Yaskawa INFORM job: X2_103(30,90)_V2.JBI

/JOB
//NAME X2_103(30,90)_V2
//POS
///NPOS 560,560,560,21,0,0
///TOOL 0
///POSTYPE PULSE
///PULSE
C00000=3271,-119374,-120746,-350,28955,423
C00001=-140235,-154096,-123138,2898,12995,-682
C00002=-200060,-156091,-101839,15852,59862,-55345
C00003=-224418,-53337,-27640,-2214,78542,-35069
C00004=-224438,-48029,-16239,-2251,74255,-34999
C00005=-222894,-44537,-9885,-2258,72183,-34438
C00006=-222281,-43062,-7261,-2261,71343,-34215
C00007=-219801,-41941,-6326,-2232,71409,-33379
C00008=-219801,-41166,-4818,-2238,70878,-33369
C00009=-219801,-41941,-6326,-2232,71409,-33379
C00010=-221729,-42672,-6756,-2255,71247,-34028
C00011=-221606,-41865,-5246,-2258,70739,-33978
C00012=-220679,-41360,-4730,-2248,70703,-33665
C00013=-221121,-41526,-4828,-2254,70667,-33813
C00014=-222894,-44537,-9885,-2258,72183,-34438
C00015=-224438,-48029,-16239,-2251,74255,-34999
C00016=-224391,-58970,-41460,-2187,84149,-35159
C00017=-200676,-32931,-16327,-317,66839,-14722
C00018=-188142,840,19554,1763,51642,-2042
C00019=-188000,8373,29094,1754,49640,-2018
C00020=-187946,11534,33150,1753,48768,-2011
C00021=-187952,12994,36316,1788,47570,-2035
C00022=-187946,11534,33150,1753,48768,-2011
C00023=-185876,12386,34874,-2226,48172,1956
C00024=-184694,15261,37512,-5775,48427,5518
C00025=-187925,12395,34881,1761,48145,-2013
C00026=-187893,12200,34611,1745,48210,-1998
C00027=-186938,14194,36446,1333,48088,-1587
C00028=-187893,12200,34611,1745,48210,-1998
C00029=-187946,9000,30501,1745,49095,-2005
C00030=-188087,1386,20853,1753,51122,-2028
C00031=-181732,-4900,4438,-770,58086,538
C00032=-174031,-1565,13615,-3944,54266,3743
C00033=-174319,5596,22673,-3924,52362,3698
C00034=-174429,8580,26495,-3922,51540,3684
C00035=-174433,9836,29416,-3983,50391,3728
C00036=-174429,8580,26495,-3922,51540,3684
C00037=-171116,10926,29585,-10065,52158,10061
C00038=-171940,12922,31394,-9974,52039,9961
C00039=-174482,9161,28010,-3935,50905,3687
C00040=-174468,9090,27852,-3937,50966,3690
C00041=-173667,11408,29941,-4272,50912,4030
C00042=-174468,9090,27852,-3937,50966,3690
C00043=-174358,6073,23987,-3937,51798,3704
C00044=-174072,-1158,14840,-3954,53720,3748
C00045=-173402,-7254,1011,1102,53334,3695
C00046=-173128,11811,16147,-4053,59614,3903
C00047=-173414,18752,25429,-4036,57459,3871
C00048=-173524,21666,29357,-4035,56536,3862
C00049=-173528,22669,32063,-4087,55389,3904
C00050=-173524,21666,29357,-4035,56536,3862
C00051=-172107,23003,31802,-6738,56186,6669
C00052=-172603,25249,33980,-7141,56088,7090
C00053=-173534,22315,31141,-4067,55773,3887
C00054=-175831,15088,24311,-3157,56159,2953
C00055=-175704,15840,26859,-3250,54984,3039
C00056=-174934,18176,29047,-3559,54871,3355
C00057=-175704,15840,26859,-3250,54984,3039
C00058=-175831,15088,24311,-3157,56159,2953
C00059=-173128,11811,16147,-4053,59614,3903
C00060=-158515,-47697,-14966,-51437,42315,-4350
C00061=-160188,-28820,10706,-61150,35121,-4094
C00062=-160938,-21306,18376,-62092,34254,-3699
C00063=-161219,-18227,21598,-62564,33894,-3488
C00064=-160407,-15938,23271,-62524,34443,-3379
C00065=-161219,-18227,21598,-62564,33894,-3488
C00066=-160594,-16595,22837,-62582,34299,-3378
C00067=-160592,-14820,26146,-64075,33771,-2570
C00068=-160594,-16595,22837,-62582,34299,-3378
C00069=-158698,-15537,23539,-63423,38355,-1788
C00070=-159328,-13237,25258,-63387,39000,-1639
C00071=-161141,-18339,21498,-62573,33942,-3471
C00072=-160858,-21416,18279,-62104,34303,-3680
C00073=-160103,-28926,10617,-61167,35171,-4072
C00074=-155148,-57735,-20992,-34211,37115,-7304
C00075=-144375,-92197,-43920,10369,38826,-10763
C00076=-123336,-72493,-22760,45909,48339,-7168
C00077=-110382,-36118,14049,67828,50364,-5484
C00078=-108060,-29324,20980,68768,48684,-5556
C00079=-107188,-26521,23897,69189,48032,-5626
C00080=-107504,-24071,25534,68933,48315,-5530
C00081=-107188,-26521,23897,69189,48032,-5626
C00082=-107470,-24738,25138,69020,48257,-5582
C00083=-107461,-22674,28687,69966,47830,-6220
C00084=-107470,-24738,25138,69020,48257,-5582
C00085=-107297,-26582,23837,69168,48098,-5639
C00086=-105452,-26141,24117,69389,47026,-5331
C00087=-107297,-26582,23837,69168,48098,-5639
C00088=-108171,-29382,20923,68748,48751,-5570
C00089=-110499,-36171,13998,67809,50435,-5499
C00090=-121659,-48497,-1187,64920,67113,80
C00091=-111034,-19450,-2794,41225,71575,-4827
C00092=-95590,24468,20339,13593,66440,-13992
C00093=-94636,30658,29262,13540,64031,-13917
C00094=-94266,33287,33052,13536,63014,-13897
C00095=-94260,34102,35593,13669,61899,-14031
C00096=-94266,33287,33052,13536,63014,-13897
C00097=-94257,33804,34719,13622,62273,-13984
C00098=-93260,34925,35856,13322,61987,-13631
C00099=-94257,33804,34719,13622,62273,-13984
C00100=-93131,24579,25521,13160,62983,-13463
C00101=-93277,25237,27975,13342,61865,-13653
C00102=-93655,28227,30921,13496,61658,-13825
C00103=-93277,25237,27975,13342,61865,-13653
C00104=-93131,24579,25521,13160,62983,-13463
C00105=-94266,33287,33052,13536,63014,-13897
C00106=-94636,30658,29262,13540,64031,-13917
C00107=-95590,24468,20339,13593,66440,-13992
C00108=-97908,6855,5922,13137,61050,-15522
C00109=-95297,11242,18824,14178,60690,-14590
C00110=-94266,17792,27740,14146,58451,-14474
C00111=-93867,20555,31520,14152,57502,-14440
C00112=-93860,21684,34363,14333,56366,-14591
C00113=-93867,20555,31520,14152,57502,-14440
C00114=-93834,21021,32943,14240,56879,-14511
C00115=-92751,22112,33981,13895,56618,-14106
C00116=-93834,21021,32943,14240,56879,-14511
C00117=-93847,20969,32801,14234,56940,-14507
C00118=-94233,23977,35706,14399,56772,-14687
C00119=-93847,20969,32801,14234,56940,-14507
C00120=-94245,18170,28975,14223,57899,-14539
C00121=-95277,11545,19966,14246,60155,-14652
C00122=-94527,-29265,-13111,13981,59468,-14364
C00123=-81565,-27458,3058,10852,48627,-10401
C00124=-80654,-20498,11026,10706,47205,-10165
C00125=-80308,-17644,14351,10663,46591,-10083
C00126=-80298,-16160,17342,10850,45531,-10203
C00127=-80308,-17644,14351,10663,46591,-10083
C00128=-80310,-16770,15973,10760,46052,-10147
C00129=-78983,-15416,16967,10190,45971,-9563
C00130=-80310,-16770,15973,10760,46052,-10147
C00131=-80369,-16920,15767,10776,46108,-10166
C00132=-81126,-14569,17524,11066,46330,-10477
C00133=-80369,-16920,15767,10776,46108,-10166
C00134=-80716,-19796,12409,10816,46731,-10247
C00135=-81629,-26799,4373,10955,48172,-10481
C00136=-81629,-36021,-16280,9851,56019,-9665
C00137=-81629,-36021,-16280,9851,56019,-9665
C00138=-81018,-22368,15352,11535,43694,-10760
C00139=-82220,-12770,25334,12334,42674,-11455
C00140=-82220,-11619,27495,12508,41954,-11560
C00141=-82220,-11847,27069,12473,42095,-11540
C00142=-82921,-9583,28807,12754,42287,-11838
C00143=-82839,-9854,28597,12721,42264,-11802
C00144=-82839,-10288,27783,12653,42536,-11762
C00145=-82987,-9794,28166,12713,42576,-11825
C00146=-82987,-9519,28676,12758,42403,-11847
C00147=-82987,-9667,28396,12734,42496,-11833
C00148=-83090,-9325,28661,12774,42522,-11877
C00149=-82753,-11045,26659,12547,42813,-11678
C00150=-119816,-37733,5380,24735,50291,-26788
C00151=-118732,-28444,14282,24759,49358,-26561
C00152=-118732,-27369,16233,24992,48768,-26724
C00153=-118733,-27539,15928,24955,48860,-26698
C00154=-118781,-24844,17728,24865,49124,-26646
C00155=-118771,-25424,17338,24885,49069,-26656
C00156=-118771,-25846,16569,24792,49302,-26592
C00157=-118785,-25058,17100,24768,49376,-26577
C00158=-118785,-24858,17464,24811,49265,-26606
C00159=-118785,-24952,17291,24791,49318,-26592
C00160=-118793,-24494,17602,24777,49360,-26584
C00161=-118763,-26610,15508,24704,49533,-26524
C00162=-155285,-26516,12514,28456,62214,-38311
C00163=-152438,-18325,21238,28659,60298,-37701
C00164=-152440,-17188,23354,28851,59667,-37879
C00165=-152440,-17414,22937,28813,59790,-37845
C00166=-151830,-15112,24623,28749,59726,-37617
C00167=-151901,-15387,24419,28758,59733,-37642
C00168=-151901,-15814,23624,28683,59971,-37576
C00169=-151771,-15314,23995,28670,59956,-37527
C00170=-151769,-15045,24491,28721,59807,-37565
C00171=-151767,-15191,24216,28696,59889,-37542
C00172=-151679,-14843,24474,28688,59877,-37510
C00173=-151971,-16573,22523,28616,60244,-37525
C00174=-150216,-29821,9901,28279,60539,-36735
C00175=-129415,-40611,3678,-20754,45854,21846
C00176=-132229,-30881,12703,-20034,44681,20835
C00177=-132233,-29758,14737,-20264,44044,20982
C00178=-132233,-29979,14337,-20217,44170,20950
C00179=-131980,-27625,15872,-20209,44476,20997
C00180=-132007,-27902,15689,-20213,44443,20995
C00181=-132009,-28325,14925,-20124,44681,20937
C00182=-131956,-27813,15263,-20122,44745,20946
C00183=-131946,-27551,15737,-20184,44594,20990
C00184=-131944,-27692,15476,-20156,44679,20973
C00185=-131906,-27334,15713,-20158,44724,20979
C00186=-132026,-29082,13878,-20039,44914,20879
C00187=-163713,-23600,14498,-6442,42405,6672
C00188=-163955,-12441,25582,-6447,41301,6644
C00189=-163960,-11291,27745,-6536,40565,6698
C00190=-163959,-11518,27319,-6518,40711,6685
C00191=-163182,-9327,29005,-6883,40857,7042
C00192=-163270,-9587,28803,-6845,40841,7005
C00193=-163272,-10021,27989,-6806,41118,6980
C00194=-163107,-9544,28360,-6883,41148,7055
C00195=-163099,-9280,28861,-6910,40971,7077
C00196=-163096,-9426,28582,-6901,41068,7072
C00197=-162981,-9093,28842,-6958,41088,7124
C00198=-163354,-10779,26863,-6731,41408,6921
C00199=-188135,19294,49745,5326,42598,-4607
C00200=-187094,34022,67542,5190,39163,-4331
C00201=-187099,35860,70809,5317,38103,-4403
C00202=-187098,35492,70157,5290,38315,-4390
C00203=-186242,38033,72879,4886,37897,-3996
C00204=-186340,37725,72546,4929,37948,-4039
C00205=-186342,37004,71278,4886,38357,-4015
C00206=-186159,37561,71878,4800,38266,-3932
C00207=-186153,37998,72654,4828,38007,-3942
C00208=-186151,37748,72215,4808,38149,-3930
C00209=-186023,38140,72638,4745,38082,-3873
C00210=-186437,35890,69530,4881,38858,-4029
C00211=-129415,-40611,3678,-20754,45854,21846
C00212=-138780,-33942,5724,-2673,47750,14957
C00213=-138299,-28814,11765,-2887,46684,15190
C00214=-170916,-2456,31220,8184,49299,1571
C00215=-171700,-5880,26786,8312,50334,1335
C00216=-135165,-49074,-6503,-3925,47635,16482
C00217=-161317,-13185,16777,20608,75826,-36642
C00218=-153104,-7651,23168,21233,72811,-34265
C00219=-161765,5352,36611,20811,73420,-37224
C00220=-160783,10050,41998,20985,72342,-37069
C00221=-152064,364,33603,21550,70406,-34339
C00222=-119342,-11748,23912,21569,62025,-23940
C00223=-119305,-17523,16883,21319,63284,-23678
C00224=-135165,-49074,-6503,-3925,47635,16482
C00225=-129415,-40611,3678,-20754,45854,21846
C00226=-171396,-8104,23990,8148,50880,1508
C00227=-170916,-2456,31220,8184,49299,1571
C00228=-192273,66939,103329,16264,43671,-8278
C00229=-192892,57382,88980,15390,47553,-7857
C00230=-135165,-49074,-6503,-3925,47635,16482
C00231=-161317,-13185,16777,20608,75826,-36642
C00232=-119244,-24750,9342,21153,64138,-23490
C00233=-119300,-17410,17676,21394,62882,-23755
C00234=-119342,-11748,23912,21569,62025,-23940
C00235=-84728,5286,37848,17156,54382,-11867
C00236=-85414,851,32833,17125,55288,-11988
C00237=-135165,-49074,-6503,-3925,47635,16482
C00238=-129360,-40332,3441,-20673,46138,21804
C00239=-138676,-33640,5524,-2697,48031,14993
C00240=-138191,-28354,11811,-2916,46896,15229
C00241=-170671,-2058,31280,8087,49442,1685
C00242=-171477,-5655,26582,8215,50551,1445
C00243=-135070,-48777,-6734,-3939,47933,16510
C00244=-161130,-12883,16630,20602,76011,-36544
C00245=-160264,65,29057,20749,74872,-36438
C00246=-160370,4102,35147,20897,73330,-36750
C00247=-164437,-245,35228,27243,65873,-40715
C00248=-155010,-10107,27390,27339,62790,-37870
C00249=-119242,-19669,19375,23179,54823,-25430
C00250=-119312,-17166,16760,21274,63528,-23633
C00251=-135070,-48777,-6734,-3939,47933,16510
C00252=-129360,-40332,3441,-20673,46138,21804
C00253=-171172,-7872,23791,8052,51098,1618
C00254=-170796,-1768,31531,8129,49447,1635
C00255=-192018,67019,103005,16124,43862,-8129
C00256=-192674,57393,88583,15275,47758,-7731
C00257=-135070,-48777,-6734,-3939,47933,16510
C00258=-161130,-12883,16630,20602,76011,-36544
C00259=-119252,-24388,9211,21109,64389,-23445
C00260=-119307,-17059,17547,21348,63127,-23710
C00261=-115642,-27884,15061,20579,45940,-25049
C00262=-76385,-6634,29757,2420,43140,-7452
C00263=-85568,1158,32706,17108,55544,-12007
C00264=-135070,-48777,-6734,-3939,47933,16510
C00265=-81018,-22368,15352,11535,43694,-10760
C00266=-90296,-130023,-32460,1589,43332,9709
C00267=-104076,-127604,-31640,1030,44224,5222
C00268=-104076,-125902,-29753,1035,43937,5219
C00269=-104076,-127604,-31640,1030,44224,5222
C00270=-75365,-129597,-31294,2148,42603,14582
C00271=-79043,-127585,-29221,2027,42422,13375
C00272=-98067,-126626,-29482,1288,43342,7171
C00273=-91643,-127131,-29393,1548,42950,9262
C00274=-91643,-133346,-36144,1521,43911,9279
C00275=-90543,-138207,-41193,1547,44504,9649
C00276=-97075,-139435,-37667,8780,42441,4238
C00277=-97192,-133417,-31365,8906,41673,4121
C00278=-82208,-129108,-27879,9651,40633,8927
C00279=-74453,-129099,-27873,9918,40030,11450
C00280=-77506,-125561,-24368,25333,36038,-6444
C00281=-97622,-127372,-24807,30901,38923,-18802
C00282=-97583,-132582,-30437,30417,39596,-18508
C00283=-96835,-139510,-37769,-4213,44951,10151
C00284=-96981,-133489,-31463,-4286,44162,10144
C00285=-62865,-129479,-28052,-642,44803,20513
C00286=-78696,-129496,-28185,-2375,44685,15709
C00287=-65731,-129649,-28076,-960,44711,19643
C00288=-97517,-133431,-31347,-4343,44102,9982
C00289=-97378,-139453,-37655,-4269,44892,9987
C00290=-122537,-139380,-37444,-6562,43692,2224
C00291=-122537,-133356,-31132,-6657,42908,2284
C00292=-123909,-129354,-27957,-6756,42937,1849
C00293=-136767,-129599,-28086,-7733,42151,-2168
C00294=-136042,-129584,-28096,-7681,42205,-1941
C00295=-122565,-109770,-4675,-55538,56258,9899
C00296=-122572,-114852,-10615,-54984,56869,9434
C00297=-218346,-133610,-69952,-6045,59781,-31164
C00298=-223401,-45840,-13156,-5364,69548,-33408
C00299=-222109,-41719,-6333,-5495,67560,-32869
C00300=-220997,-38818,-2909,-5568,67023,-32457
C00301=-222242,-31345,1911,-5480,67806,-32926
C00302=-220920,-39606,-2024,-7766,59138,-23574
C00303=-220403,-51511,-7368,-9623,49930,-15864
C00304=-221089,-58034,-14727,-9279,51017,-16249
C00305=-225149,-36583,-7538,-3060,79587,-35998
C00306=-223778,-33707,-1346,-2977,77308,-35487
C00307=-222503,-31636,1503,-2884,76662,-35050
C00308=-221605,-36907,-1779,-2822,76007,-34739
C00309=-217292,-55512,-12105,-2514,72937,-33253
C00310=-219328,-56399,-14375,-2668,73818,-33940
C00311=-221046,-59770,-20585,-2780,75851,-34551
C00312=-232710,-104201,-36509,-3988,62401,-37975
C00313=-229171,-99745,-30242,-3753,60982,-36787
C00314=-225249,-97366,-27202,-3443,60481,-35515
C00315=-159716,-121406,-28671,3019,49335,-15001
C00316=-178146,-119749,-28353,3122,51852,-21289
C00317=-201053,-127933,-48461,1469,67517,-27836
C00318=-218346,-133610,-69952,-6045,59781,-31164
C00319=-155907,-158824,-62139,3482,48253,-13777
C00320=-122507,-139290,-37311,6932,43923,-3746
C00321=-122509,-133268,-31001,7032,43139,-3809
C00322=-129091,-129141,-27877,6412,43686,-5823
C00323=-103454,-129456,-28220,8487,42206,2149
C00324=-122587,-133369,-31211,7015,43220,-3827
C00325=-122586,-139389,-37517,6916,44002,-3765
C00326=-178554,-156416,-68062,-1714,49894,-19175
C00327=-213759,-120199,-38675,-7265,47820,-28777
C00328=-208805,-113975,-32275,-7533,47440,-26995
C00329=-203457,-110659,-29180,-7720,47634,-25130
C00330=-226422,-78834,-22033,-5752,57916,-33897
C00331=-229015,-79900,-24597,-5554,58778,-34856
C00332=-231182,-84689,-31124,-5352,60195,-35689
C00333=-212528,-138829,-62774,-5865,50017,-28724
C00334=-155907,-158824,-62139,3482,48253,-13777
C00335=-121094,-142626,-31574,-10098,25521,4701
C00336=-121096,-137018,-25859,-10336,24895,4818
C00337=-164582,-134101,-22446,3427,23155,-15265
C00338=-111553,-133057,-22885,-12578,25881,8893
C00339=-110779,-133123,-22850,-12777,25898,9232
C00340=-112921,-147420,-34515,-12366,25547,8360
C00341=-112921,-149481,-36511,-12292,25712,8323
C00342=-97228,-139073,-37279,8780,42400,4184
C00343=-97344,-133056,-30967,8907,41624,4066
C00344=-78012,-130084,-28544,9824,40218,10278
C00345=-81788,-129487,-28074,9683,40529,9053
C00346=-82179,-129411,-27981,9668,40535,8924
C00347=-74028,-129648,-28142,9954,39883,11573
C00348=-97200,-133072,-30998,8914,41625,4113
C00349=-97082,-139088,-37310,8787,42400,4232
C00350=-94488,-144762,-30508,4018,22458,6207
C00351=-94506,-139089,-24810,4127,21868,6148
C00352=-109156,-134471,-22107,8848,23225,-653
C00353=-92905,-135418,-22246,3518,22151,6937
C00354=-86752,-134662,-22676,6773,23151,2299
C00355=-94482,-131728,-17188,50151,23285,-24299
C00356=-94477,-136650,-22327,49039,23703,-23756
C00357=-194092,-153326,-35489,27084,38346,-44238
C00358=-219173,-157061,-72685,-6819,49419,-30815
C00359=-224435,-92754,-33276,-5864,57810,-33193
C00360=-222031,-87567,-26717,-6069,56604,-32279
C00361=-219894,-84961,-24547,-6166,56749,-31533
C00362=-220391,-83143,-23447,-6127,56973,-31723
C00363=-220808,-82168,-23250,-6081,57322,-31890
C00364=-221831,-79477,-22462,-5978,58145,-32293
C00365=-223925,-82065,-24949,-5866,58209,-33035
C00366=-226120,-87049,-31520,-5671,59544,-33877
C00367=-225186,-114904,-34894,11668,45054,-37894
C00368=-216822,-109183,-29035,10924,43485,-34913
C00369=-213756,-104039,-26334,10373,44131,-33658
C00370=-227756,-76443,-19510,10264,55464,-37669
C00371=-223895,-83934,-20074,8254,42953,-29929
C00372=-217578,-99941,-27704,3828,33118,-22325
C00373=-218675,-113856,-37596,3440,30409,-21358
C00374=-233993,-86215,-29007,10771,66078,-41518
C00375=-229810,-82565,-23340,11182,63991,-40325
C00376=-227706,-76286,-19097,11255,64337,-39587
C00377=-202149,-109903,-26387,14167,48571,-32832
C00378=-202051,-109942,-26389,14173,48540,-32803
C00379=-202051,-128717,-48625,13393,52466,-32246
C00380=-202051,-134657,-55264,13217,53473,-32112
C00381=-117234,-149912,-54866,6773,48847,-5879
C00382=-121099,-142746,-31792,-10070,25592,4686
C00383=-121100,-137139,-26082,-10306,24969,4802
C00384=-141051,-133855,-23509,-4396,24027,-4240
C00385=-121100,-133451,-23236,-10248,25112,4773
C00386=-121096,-137018,-25859,-10336,24895,4818
C00387=-121094,-142626,-31574,-10098,25521,4701
C00388=-123662,-145584,-42609,-8092,33284,3232
C00389=-230686,-106057,-33987,11415,49598,-39384
C00390=-224512,-100771,-28076,11039,47987,-37279
C00391=-205796,-94439,-26049,241,49435,-28150
C00392=-216777,-58757,-13663,-3179,61810,-31293
C00393=-233092,-64153,-16123,10229,60240,-39150
C00394=-236163,-68268,-22160,10284,62176,-40071
C00395=-236095,-83218,-48894,9648,70813,-39304
C00396=-106397,-55795,3096,63565,21817,17186
C00397=-106632,-48373,10599,65478,21584,16223
C00398=-106548,-45729,13184,65997,21437,15992
C00399=-103258,-44886,13759,64702,19643,17243
C00400=-95899,-43443,14256,59303,15873,21157
C00401=-118505,-22556,31998,69880,50592,992
C00402=-120549,-21950,32011,69247,53773,-244
C00403=-109887,-57295,-6780,52006,39852,10060
C00404=-88953,-54538,-6858,-3495,30900,36178
C00405=-87457,-47486,-1790,-16888,35291,41492
C00406=-88117,-45133,941,-16673,34715,41263
C00407=-112697,-47495,6210,47940,30588,13914
C00408=-106422,-46154,7077,44887,27834,16652
C00409=-122247,-33138,27647,79444,43496,6604
C00410=-123052,-35890,24633,78754,44065,6817
C00411=-125208,-43152,16784,77075,45600,7305
C00412=-136500,-67051,-4345,73514,52458,6539
C00413=-180716,-92339,-35753,46571,44741,-29909
C00414=-181887,-65932,-22068,22787,28646,-43428
C00415=-164154,-32069,4835,-4706,35458,-29947
C00416=-162862,-25243,12769,-5829,34168,-29145
C00417=-162318,-22407,15975,-6313,33693,-28802
C00418=-164433,-20534,17116,-4694,33821,-29993
C00419=-169618,-16577,21269,848,31718,-33215
C00420=-148668,-7920,37360,-58299,39489,-2391
C00421=-148264,-10930,34029,-57819,39984,-2589
C00422=-147210,-18873,24978,-56466,41391,-3180
C00423=-153881,-52361,-9825,-51389,40377,-7407
C00424=-195451,-44212,-13367,33096,44702,-59640
C00425=-188165,-11987,14443,28697,52592,-54038
C00426=-185681,-7933,20770,28676,50175,-53635
C00427=-185046,-6113,23212,28716,49467,-53563
C00428=-170951,-24048,16105,-1564,23385,-43494
C00429=-175189,-18557,20056,3862,23831,-46738
C00430=-164622,-16739,33688,-78292,16289,-16544
C00431=-164679,-19923,29950,-76041,16420,-17596
C00432=-165032,-27921,20991,-71332,16638,-19843
C00433=-159893,-54487,-7231,-63606,21243,-22673
C00434=-154676,-47992,-9690,-48263,49204,2905
C00435=-193585,-9261,11754,-11559,55982,16808
C00436=-194745,-2712,20199,-11444,54025,16555
C00437=-194872,621,24646,-11550,53002,16618
C00438=-184827,19619,41586,-14742,53935,20630
C00439=-184159,21046,43063,-14423,52970,15772
C00440=-184002,17429,38335,-14281,54014,15688
C00441=-182921,10224,28561,-14216,56443,15793
C00442=-177083,-111,8338,-7845,50349,39492
C00443=-178532,5317,16012,-7278,48297,39013
C00444=-179015,7475,19264,-7110,47370,38866
C00445=-178120,9780,21301,-7616,47383,39270
C00446=-171533,31347,41892,-11486,46586,42364
C00447=-173045,27120,40896,-5889,38045,43816
C00448=-172668,24060,36713,-6048,39069,43937
C00449=-171398,17656,27538,-6677,41509,44399
C00450=-161344,12362,8811,-26436,45100,67481
C00451=-163521,18252,18448,-26269,41792,67367
C00452=-161897,26643,30849,-29661,32619,71760
C00453=-161203,20965,26512,-31560,29825,74587
C00454=-161149,7456,11537,-29677,31816,73606
C00455=-175227,6351,5531,-3063,39549,38971
C00456=-186824,8866,15973,21206,34489,4565
C00457=-186762,16678,24474,21808,33336,4242
C00458=-186659,19688,27148,21766,33216,4273
C00459=-187823,20782,34277,25409,30033,2285
C00460=-189098,23597,36861,27884,33394,5871
C00461=-189065,20396,33165,27418,33944,6127
C00462=-189139,12249,23817,26457,35372,6645
C00463=-201440,-17736,15052,46372,30187,-8745
C00464=-200958,-18911,21572,51828,25568,-12457
C00465=-200198,-11285,28867,52326,24814,-12587
C00466=-199904,-8230,31793,52545,24518,-12649
C00467=-201573,-3368,42099,60720,23241,-16913
C00468=-203007,-101,44904,57709,26762,-11216
C00469=-203186,-3827,40838,56798,27185,-10789
C00470=-203962,-12064,32256,55427,28201,-10233
C00471=-200938,-30348,-961,41051,31198,-6989
C00472=-160850,-63419,-43720,34430,57956,-16775
C00473=-110095,-57810,-32372,23714,72198,-38531
C00474=-93378,-40488,-5092,23425,60303,-34603
C00475=-90533,-35882,1051,23375,58234,-33930
C00476=-89429,-33691,4119,23410,57240,-33713
C00477=-95242,-8050,22330,23694,60617,-35274
C00478=-95768,-6357,23797,23918,59729,-30488
C00479=-96526,-9092,20324,23849,60611,-30591
C00480=-98793,-14030,13298,23755,62879,-30983
C00481=-94098,-24836,421,24737,48725,-53543
C00482=-91650,-20510,6675,24341,46535,-52972
C00483=-90508,-18507,9931,24234,45316,-52749
C00484=-95414,7977,31078,26011,47297,-54577
C00485=-94573,3656,30653,27510,37763,-58721
C00486=-95383,1086,27130,27491,38776,-58811
C00487=-97471,-4004,19715,27585,41178,-59115
C00488=-94564,2818,10716,38987,45684,-75599
C00489=-92587,6675,17082,39222,43275,-75644
C00490=-91561,8164,19761,39289,42122,-75622
C00491=-92468,13395,24417,39885,42394,-76048
C00492=-93952,23755,34118,41077,42576,-76882
C00493=-90590,7329,26151,50031,24200,-87071
C00494=-96600,-9343,13340,55774,27143,-90423
C00495=-97074,-7723,20735,33897,25089,-35230
C00496=-95399,-742,27921,33089,23755,-34646
C00497=-94753,2002,30741,32759,23241,-34410
C00498=-94210,4250,38659,37485,19954,-36607
C00499=-92176,4748,39092,25289,19678,-35891
C00500=-92831,1779,35666,25549,20393,-36102
C00501=-94452,-5624,27606,26438,21912,-36738
C00502=-98858,-50483,238,51569,18835,-43949
C00503=-96204,-39490,13375,55375,15987,-45282
C00504=-95397,-37131,15438,54750,15537,-44853
C00505=-94515,-33287,24483,66247,13200,-49976
C00506=-91286,-32749,24823,46845,10625,-45650
C00507=-92274,-35440,22191,47758,11230,-46248
C00508=-94786,-42118,16150,50717,12576,-48060
C00509=-89658,-85206,-39306,19320,21137,-32731
C00510=-106882,-134348,-55470,2817,27003,-12032
C00511=-115899,-155260,-61631,-2537,28837,-4647
C00512=-121094,-142626,-31574,-10098,25521,4701
C00513=-121096,-137018,-25859,-10336,24895,4818
C00514=-164582,-134101,-22446,3427,23155,-15265
C00515=-111553,-133057,-22885,-12578,25881,8893
C00516=-110779,-133123,-22850,-12777,25898,9232
C00517=-112921,-147420,-34515,-12366,25547,8360
C00518=-112921,-149481,-36511,-12292,25712,8323
C00519=-97227,-139073,-37279,8780,42400,4185
C00520=-97341,-133056,-30967,8908,41624,4067
C00521=-78007,-130084,-28544,9824,40218,10280
C00522=-81785,-129487,-28074,9683,40529,9054
C00523=-82177,-129411,-27981,9668,40535,8924
C00524=-74024,-129648,-28142,9954,39882,11575
C00525=-97198,-133072,-30998,8914,41625,4113
C00526=-97081,-139088,-37310,8787,42400,4233
C00527=-94488,-144762,-30508,4018,22458,6207
C00528=-94506,-139089,-24810,4127,21868,6148
C00529=-109156,-134471,-22107,8848,23225,-653
C00530=-92905,-135418,-22246,3518,22151,6937
C00531=-86752,-134662,-22676,6773,23151,2299
C00532=-94482,-131728,-17188,50151,23285,-24299
C00533=-94477,-136650,-22327,49039,23703,-23756
C00534=-194092,-153326,-35489,27084,38346,-44238
C00535=-219173,-157061,-72685,-6819,49419,-30815
C00536=-224435,-92754,-33276,-5864,57810,-33193
C00537=-222031,-87567,-26717,-6069,56604,-32279
C00538=-219894,-84961,-24547,-6166,56749,-31533
C00539=-220391,-83143,-23447,-6127,56973,-31723
C00540=-220808,-82168,-23250,-6081,57322,-31890
C00541=-221831,-79477,-22462,-5978,58145,-32293
C00542=-223925,-82065,-24949,-5866,58209,-33035
C00543=-226120,-87049,-31520,-5671,59544,-33877
C00544=-225186,-114904,-34894,11668,45054,-37894
C00545=-216822,-109183,-29035,10924,43485,-34913
C00546=-213756,-104039,-26334,10373,44131,-33658
C00547=-227756,-76443,-19510,10264,55464,-37669
C00548=-223895,-83934,-20074,8254,42953,-29929
C00549=-217578,-99941,-27704,3828,33118,-22325
C00550=-218675,-113856,-37596,3440,30409,-21358
C00551=-233993,-86215,-29007,10771,66078,-41518
C00552=-229810,-82565,-23340,11182,63991,-40325
C00553=-227706,-76286,-19097,11255,64337,-39587
C00554=-202149,-109903,-26387,14167,48571,-32832
C00555=-202051,-109942,-26389,14173,48540,-32803
C00556=-202051,-128717,-48625,13393,52466,-32246
C00557=-202051,-134657,-55264,13217,53473,-32112
C00558=-134221,-121505,-102040,30238,34212,-41263
C00559=3271,-119374,-120746,-350,28955,423
BC00000=132383,666204,1075229
BC00001=261940,799209,1050994
BC00002=248524,1011966,1050994
BC00003=202466,1017054,1075175
BC00004=202466,1017054,1075175
BC00005=202466,1017054,1075175
BC00006=202466,1017054,1075175
BC00007=202466,1017054,1075175
BC00008=202466,1017054,1075175
BC00009=202466,1017054,1075175
BC00010=202466,1017054,1075175
BC00011=202466,1017054,1075175
BC00012=202466,1017054,1075175
BC00013=202466,1017054,1075175
BC00014=202466,1017054,1075175
BC00015=202466,1017054,1075175
BC00016=202466,1017054,1075175
BC00017=230796,978668,1056603
BC00018=250273,952277,1043835
BC00019=250273,952277,1043835
BC00020=250273,952277,1043835
BC00021=250273,952277,1043835
BC00022=250273,952277,1043835
BC00023=250273,952277,1043835
BC00024=250273,952277,1043832
BC00025=250273,952277,1043835
BC00026=250273,952277,1043835
BC00027=250273,952277,1043835
BC00028=250273,952277,1043835
BC00029=250273,952277,1043835
BC00030=250273,952277,1043835
BC00031=239388,961471,1057989
BC00032=226170,972635,1075175
BC00033=226170,972635,1075175
BC00034=226170,972635,1075175
BC00035=226170,972635,1075175
BC00036=226170,972635,1075175
BC00037=226170,972635,1075175
BC00038=226170,972635,1075175
BC00039=226170,972635,1075175
BC00040=226170,972635,1075175
BC00041=226170,972635,1075175
BC00042=226170,972635,1075175
BC00043=226170,972635,1075175
BC00044=226170,972635,1075175
BC00045=234013,971063,1075175
BC00046=236865,970491,1075175
BC00047=236865,970491,1075175
BC00048=236865,970491,1075175
BC00049=236865,970491,1075175
BC00050=236865,970491,1075175
BC00051=236865,970491,1075175
BC00052=236865,970491,1075175
BC00053=236865,970491,1075175
BC00054=236865,970491,1075175
BC00055=236865,970491,1075175
BC00056=236865,970491,1075175
BC00057=236865,970491,1075175
BC00058=236865,970491,1075175
BC00059=236865,970491,1075175
BC00060=241076,1045232,1015466
BC00061=241654,1055491,1007270
BC00062=241654,1055491,1007270
BC00063=241654,1055491,1007270
BC00064=241654,1055491,1007270
BC00065=241654,1055491,1007270
BC00066=241654,1055491,1007270
BC00067=241654,1055491,1007270
BC00068=241654,1055491,1007270
BC00069=241654,1055491,1007270
BC00070=241654,1055491,1007270
BC00071=241654,1055491,1007270
BC00072=241654,1055491,1007270
BC00073=241654,1055491,1007270
BC00074=243378,1058693,1018091
BC00075=246825,1065098,1039733
BC00076=250380,1071704,1062053
BC00077=248912,1056159,1048449
BC00078=248912,1056159,1048449
BC00079=248912,1056159,1048449
BC00080=248912,1056159,1048449
BC00081=248912,1056159,1048449
BC00082=248912,1056159,1048449
BC00083=248912,1056159,1048449
BC00084=248912,1056159,1048449
BC00085=248912,1056159,1048449
BC00086=248912,1056159,1048449
BC00087=248912,1056159,1048449
BC00088=248912,1056159,1048449
BC00089=248912,1056159,1048449
BC00090=248912,1056159,1060963
BC00091=253480,996710,1046754
BC00092=259276,921290,1028729
BC00093=259276,921290,1028729
BC00094=259276,921290,1028729
BC00095=259276,921290,1028729
BC00096=259276,921290,1028729
BC00097=259276,921290,1028729
BC00098=259276,921290,1028729
BC00099=259276,921290,1028729
BC00100=259276,921290,1028729
BC00101=259276,921290,1028729
BC00102=259276,921290,1028729
BC00103=259276,921290,1028729
BC00104=259276,921290,1028729
BC00105=259276,921290,1028729
BC00106=259276,921290,1028729
BC00107=259276,921290,1028729
BC00108=261148,922509,1033111
BC00109=264517,924704,1040999
BC00110=264517,924704,1040999
BC00111=264517,924704,1040999
BC00112=264517,924704,1040999
BC00113=264517,924704,1040999
BC00114=264517,924704,1040999
BC00115=264517,924704,1040999
BC00116=264517,924704,1040999
BC00117=264517,924704,1040999
BC00118=264517,924704,1040999
BC00119=264517,924704,1040999
BC00120=264517,924704,1040999
BC00121=264517,924704,1040999
BC00122=260067,934845,1062644
BC00123=257490,940717,1075175
BC00124=257490,940717,1075175
BC00125=257490,940717,1075175
BC00126=257490,940717,1075175
BC00127=257490,940717,1075175
BC00128=257490,940717,1075175
BC00129=257490,940717,1075175
BC00130=257490,940717,1075175
BC00131=257490,940717,1075175
BC00132=257490,940717,1075175
BC00133=257490,940717,1075175
BC00134=257490,940717,1075175
BC00135=257490,940717,1075175
BC00136=257490,940717,1075175
BC00137=257490,879918,1075175
BC00138=257490,879918,1075175
BC00139=257490,879919,1075172
BC00140=257490,879919,1075172
BC00141=257490,879919,1075172
BC00142=257490,879919,1075172
BC00143=257490,879919,1075172
BC00144=257490,879919,1075172
BC00145=257490,879919,1075172
BC00146=257490,879919,1075172
BC00147=257490,879919,1075172
BC00148=257490,879919,1075172
BC00149=257490,879919,1075172
BC00150=257490,879918,1075175
BC00151=257490,879919,1075172
BC00152=257490,879919,1075172
BC00153=257490,879919,1075172
BC00154=257490,879919,1075172
BC00155=257490,879919,1075172
BC00156=257490,879919,1075172
BC00157=257490,879919,1075172
BC00158=257490,879919,1075172
BC00159=257490,879919,1075172
BC00160=257490,879919,1075172
BC00161=257490,879919,1075172
BC00162=257490,879918,1075175
BC00163=257490,879919,1075172
BC00164=257490,879919,1075172
BC00165=257490,879919,1075172
BC00166=257490,879919,1075172
BC00167=257490,879919,1075172
BC00168=257490,879919,1075172
BC00169=257490,879919,1075172
BC00170=257490,879919,1075172
BC00171=257490,879919,1075172
BC00172=257490,879919,1075172
BC00173=257490,879919,1075172
BC00174=257490,879919,1075172
BC00175=257490,879918,1075175
BC00176=257490,879919,1075172
BC00177=257490,879919,1075172
BC00178=257490,879919,1075172
BC00179=257490,879919,1075172
BC00180=257490,879919,1075172
BC00181=257490,879919,1075172
BC00182=257490,879919,1075172
BC00183=257490,879919,1075172
BC00184=257490,879919,1075172
BC00185=257490,879919,1075172
BC00186=257490,879919,1075172
BC00187=257490,879918,1075175
BC00188=257490,879919,1075172
BC00189=257490,879919,1075172
BC00190=257490,879919,1075172
BC00191=257490,879919,1075172
BC00192=257490,879919,1075172
BC00193=257490,879919,1075172
BC00194=257490,879919,1075172
BC00195=257490,879919,1075172
BC00196=257490,879919,1075172
BC00197=257490,879919,1075172
BC00198=257490,879919,1075172
BC00199=257490,879918,1075175
BC00200=257490,879919,1075172
BC00201=257490,879919,1075172
BC00202=257490,879919,1075172
BC00203=257490,879919,1075172
BC00204=257490,879919,1075172
BC00205=257490,879919,1075172
BC00206=257490,879919,1075172
BC00207=257490,879919,1075172
BC00208=257490,879919,1075172
BC00209=257490,879919,1075172
BC00210=257490,879919,1075172
BC00211=257490,879918,1075175
BC00212=257490,879919,1075172
BC00213=257490,879919,1075172
BC00214=257490,879919,1075172
BC00215=257490,879919,1075172
BC00216=257490,879919,1075172
BC00217=257490,879919,1075172
BC00218=257490,879919,1075172
BC00219=257490,879919,1075172
BC00220=257490,879919,1075172
BC00221=257490,879919,1075172
BC00222=257490,879919,1075172
BC00223=257490,879919,1075172
BC00224=257490,879919,1075172
BC00225=257490,879918,1075175
BC00226=257490,879919,1075172
BC00227=257490,879919,1075172
BC00228=257490,879919,1075172
BC00229=257490,879919,1075172
BC00230=257490,879919,1075172
BC00231=257490,879919,1075172
BC00232=257490,879919,1075172
BC00233=257490,879919,1075172
BC00234=257490,879919,1075172
BC00235=257490,879919,1075172
BC00236=257490,879919,1075172
BC00237=257490,879919,1075172
BC00238=257490,879918,1075175
BC00239=257490,879919,1075172
BC00240=257490,879919,1075172
BC00241=257490,879919,1075172
BC00242=257490,879919,1075172
BC00243=257490,879919,1075172
BC00244=257490,879919,1075172
BC00245=257490,879919,1075172
BC00246=257490,879919,1075172
BC00247=257490,879919,1075172
BC00248=257490,879919,1075172
BC00249=257490,879919,1075172
BC00250=257490,879919,1075172
BC00251=257490,879919,1075172
BC00252=257490,879918,1075175
BC00253=257490,879919,1075172
BC00254=257490,879919,1075172
BC00255=257490,879919,1075171
BC00256=257490,879919,1075172
BC00257=257490,879919,1075172
BC00258=257490,879919,1075172
BC00259=257490,879919,1075172
BC00260=257490,879919,1075172
BC00261=257490,879919,1075172
BC00262=257490,879919,1075172
BC00263=257490,879919,1075172
BC00264=257490,879919,1075172
BC00265=257490,879918,1075175
BC00266=359925,1044634,1075175
BC00267=359932,1046852,1075175
BC00268=359932,1046852,1075175
BC00269=359932,1046852,1075175
BC00270=359932,1046852,1075175
BC00271=359932,1046852,1075175
BC00272=359932,1046852,1075175
BC00273=359932,1046852,1075175
BC00274=359932,1046852,1075175
BC00275=359870,1040970,1075175
BC00276=356389,1051959,1075175
BC00277=357122,1054343,1075175
BC00278=357415,1055296,1075175
BC00279=366494,1055270,1075175
BC00280=348141,1054352,1075175
BC00281=340355,1053218,1075175
BC00282=336339,1051156,1075175
BC00283=369163,1051902,1075175
BC00284=368508,1054290,1075175
BC00285=368246,1055245,1075175
BC00286=363468,1055259,1075175
BC00287=338780,1055330,1075175
BC00288=339042,1054375,1075175
BC00289=339697,1051987,1075175
BC00290=285479,1052366,1075175
BC00291=284824,1054754,1075175
BC00292=284562,1055709,1075175
BC00293=240665,1055835,1075175
BC00294=239487,1055838,1075175
BC00295=303422,1059495,1075175
BC00296=307957,1057520,1075175
BC00297=202077,1034058,1075175
BC00298=209421,1018994,1075175
BC00299=209421,1018994,1075175
BC00300=209421,1018994,1075175
BC00301=209421,1018994,1075175
BC00302=209421,1018994,1075175
BC00303=209421,1018994,1075175
BC00304=209421,1018994,1075175
BC00305=208337,1019582,1075175
BC00306=208337,1019582,1075175
BC00307=208337,1019582,1075175
BC00308=208337,1019582,1075175
BC00309=208337,1019582,1075175
BC00310=208337,1019582,1075175
BC00311=208337,1019582,1075175
BC00312=205527,1042320,1075175
BC00313=205527,1042320,1075175
BC00314=205527,1042320,1075175
BC00315=205527,1042320,1075175
BC00316=205527,1042320,1075175
BC00317=205527,1042320,1036192
BC00318=202077,1034058,1075175
BC00319=252354,1028048,1075175
BC00320=264741,1052446,1075175
BC00321=265474,1054829,1075175
BC00322=265767,1055783,1075175
BC00323=318647,1055631,1075175
BC00324=318354,1054678,1075175
BC00325=317621,1052294,1075175
BC00326=245317,1043409,1075175
BC00327=200126,1037856,1075175
BC00328=200126,1037856,1075175
BC00329=200126,1037856,1075175
BC00330=200126,1037856,1075175
BC00331=200126,1037856,1075175
BC00332=200126,1037856,1075175
BC00333=202875,1038657,1075175
BC00334=252354,1028048,1075175
BC00335=285415,1041090,1075175
BC00336=284762,1045097,1075175
BC00337=284501,1046700,1075175
BC00338=239712,1046861,1075175
BC00339=239425,1046862,1075175
BC00340=239425,1046862,1075175
BC00341=239425,1046862,1075175
BC00342=348429,1052807,1075175
BC00343=349162,1055190,1075175
BC00344=349456,1056144,1075175
BC00345=352641,1056135,1075175
BC00346=354234,1056130,1075175
BC00347=357419,1056121,1075175
BC00348=357126,1055168,1075175
BC00349=356393,1052784,1075175
BC00350=326222,1045148,1075175
BC00351=326957,1049151,1075175
BC00352=327251,1050752,1075175
BC00353=373952,1050649,1075175
BC00354=373952,1050649,1075175
BC00355=342677,1052714,1075175
BC00356=338660,1049244,1075175
BC00357=255446,1031256,1075175
BC00358=181526,1042944,1075175
BC00359=158260,1034197,1075175
BC00360=158260,1034197,1075175
BC00361=158260,1034197,1075175
BC00362=158260,1034197,1075175
BC00363=158260,1034197,1075175
BC00364=158260,1034197,1075175
BC00365=158260,1034197,1075175
BC00366=158260,1034197,1075175
BC00367=152093,1014947,1075175
BC00368=152093,1014947,1075175
BC00369=152093,1014947,1075175
BC00370=152093,1014947,1075175
BC00371=152093,1014947,1075175
BC00372=152093,1014947,1075175
BC00373=152093,1014947,1075175
BC00374=227511,1014875,1075175
BC00375=227511,1014875,1075175
BC00376=227511,1014875,1075175
BC00377=227511,1014875,1075175
BC00378=227511,1014875,1075175
BC00379=227511,1014875,1075175
BC00380=227511,1014875,1075175
BC00381=265280,1027573,1075175
BC00382=338295,1040939,1075175
BC00383=337642,1044946,1075175
BC00384=337380,1046548,1075175
BC00385=295673,1046668,1075175
BC00386=284762,1045097,1075175
BC00387=285415,1041090,1075175
BC00388=252223,1030468,1075175
BC00389=219530,1015419,1075175
BC00390=219530,1015419,1075175
BC00391=219530,1015419,1075175
BC00392=219530,1015419,1075175
BC00393=219530,1015419,1075175
BC00394=219530,1015419,1075175
BC00395=219530,1015419,1075175
BC00396=274723,1054582,1075175
BC00397=274723,1054582,1075175
BC00398=274723,1054582,1075174
BC00399=274723,1054582,1075175
BC00400=274723,1054582,1075175
BC00401=274723,1054582,1075175
BC00402=274723,1054582,1075175
BC00403=274723,1054582,1075175
BC00404=302769,1055722,1075175
BC00405=312008,1056098,1075175
BC00406=312008,1056098,1075175
BC00407=312008,1056098,1075175
BC00408=312008,1056098,1075175
BC00409=312008,1056098,1075175
BC00410=312008,1056098,1075175
BC00411=312008,1056098,1075175
BC00412=312008,1056098,1075175
BC00413=249496,1051169,1075175
BC00414=210273,1048077,1075175
BC00415=210273,1048077,1075175
BC00416=210273,1048077,1075175
BC00417=210273,1048077,1075175
BC00418=210273,1048077,1075175
BC00419=210273,1048077,1075175
BC00420=210273,1048077,1075175
BC00421=210273,1048077,1075175
BC00422=210273,1048077,1075175
BC00423=210273,1048077,1075175
BC00424=203682,1051331,1050994
BC00425=203682,1051331,1050994
BC00426=203682,1051331,1050994
BC00427=203682,1051331,1050994
BC00428=203682,1051331,1050994
BC00429=203682,1051331,1050994
BC00430=203682,1051331,1050994
BC00431=203682,1051331,1050994
BC00432=203682,1051331,1050994
BC00433=203682,1051331,1050994
BC00434=222662,1011450,1062056
BC00435=257639,966939,1045536
BC00436=257639,966939,1045536
BC00437=257639,966939,1045536
BC00438=257639,966939,1045536
BC00439=257639,966939,1045536
BC00440=257639,966939,1045536
BC00441=257639,966939,1045536
BC00442=250000,948894,1004804
BC00443=250000,948894,1004804
BC00444=250000,948894,1004804
BC00445=250000,948894,1004804
BC00446=250000,948894,1004804
BC00447=250000,948894,1004804
BC00448=250000,948894,1004804
BC00449=250000,948894,1004804
BC00450=244323,945510,933487
BC00451=244323,945510,933487
BC00452=244323,945510,933487
BC00453=244324,945511,933483
BC00454=244324,945511,933483
BC00455=258711,950558,939336
BC00456=274206,955995,945636
BC00457=274206,955995,945636
BC00458=274206,955995,945636
BC00459=274206,955995,945636
BC00460=274206,955995,945636
BC00461=274206,955995,945636
BC00462=274206,955995,945636
BC00463=254483,964951,1031347
BC00464=249104,967393,1054722
BC00465=249104,967393,1054722
BC00466=249104,967393,1054722
BC00467=249104,967393,1054722
BC00468=249104,967393,1054722
BC00469=249104,967393,1054722
BC00470=249104,967393,1054722
BC00471=249104,967393,1054722
BC00472=260815,957267,1063697
BC00473=275794,944314,1075175
BC00474=275794,944314,1075175
BC00475=275794,944314,1075175
BC00476=275794,944314,1075175
BC00477=275794,944314,1075175
BC00478=275794,944314,1075175
BC00479=275794,944314,1075175
BC00480=275794,944314,1075175
BC00481=263746,944063,1075175
BC00482=263746,944063,1075175
BC00483=263746,944063,1075175
BC00484=263746,944063,1075175
BC00485=263746,944063,1075175
BC00486=263746,944063,1075175
BC00487=263746,944063,1075175
BC00488=235159,942078,1001811
BC00489=235159,942078,1001811
BC00490=235159,942078,1001811
BC00491=235159,942078,1001811
BC00492=235159,942078,1001811
BC00493=235159,942078,1001811
BC00494=235159,942078,1063796
BC00495=265027,925964,1060756
BC00496=265027,925964,1060756
BC00497=265027,925964,1060756
BC00498=265027,925964,1060756
BC00499=265027,925964,1060756
BC00500=265027,925964,1060756
BC00501=265027,925964,1060756
BC00502=285803,937703,1075175
BC00503=285803,937703,1075175
BC00504=285803,937703,1075175
BC00505=285803,937703,1075175
BC00506=285803,937703,1075175
BC00507=285803,937703,1075175
BC00508=285803,937703,1075175
BC00509=285803,937705,1075174
BC00510=285590,994350,1075175
BC00511=285501,1017997,1075175
BC00512=285415,1040476,1075175
BC00513=284762,1044483,1075175
BC00514=284501,1046086,1075175
BC00515=239712,1046247,1075175
BC00516=239425,1046248,1075175
BC00517=239425,1046248,1075175
BC00518=239425,1046248,1075175
BC00519=348429,1052193,1075175
BC00520=349162,1054576,1075175
BC00521=349456,1055530,1075175
BC00522=352641,1055521,1075175
BC00523=354234,1055516,1075175
BC00524=357419,1055507,1075175
BC00525=357126,1054554,1075175
BC00526=356393,1052170,1075175
BC00527=326222,1044534,1075175
BC00528=326957,1048537,1075175
BC00529=327251,1050138,1075175
BC00530=373952,1050035,1075175
BC00531=373952,1050035,1075175
BC00532=342677,1052100,1075175
BC00533=338660,1048630,1075175
BC00534=255446,1030642,1075175
BC00535=181526,1042330,1075175
BC00536=158260,1033583,1075175
BC00537=158260,1033583,1075175
BC00538=158260,1033583,1075175
BC00539=158260,1033583,1075175
BC00540=158260,1033583,1075175
BC00541=158260,1033583,1075175
BC00542=158260,1033583,1075175
BC00543=158260,1033583,1075175
BC00544=152093,1014333,1075175
BC00545=152093,1014333,1075175
BC00546=152093,1014333,1075175
BC00547=152093,1014333,1075175
BC00548=152093,1014333,1075175
BC00549=152093,1014333,1075175
BC00550=152093,1014333,1075175
BC00551=227511,1014261,1075175
BC00552=227511,1014261,1075175
BC00553=227511,1014261,1075175
BC00554=227511,1014261,1075175
BC00555=227511,1014261,1075175
BC00556=227511,1014261,1075175
BC00557=227511,1014261,1075175
BC00558=285803,876672,1075175
BC00559=132383,666204,1075229
EC00000=266052,556475
EC00001=487668,556475
EC00002=266052,556475
EC00003=266052,556475
EC00004=266052,556475
EC00005=266052,556475
EC00006=266052,556475
EC00007=266052,556475
EC00008=266052,556475
EC00009=266052,556475
EC00010=266052,556475
EC00011=266052,556475
EC00012=266052,556475
EC00013=266052,556475
EC00014=266052,556475
EC00015=266052,556475
EC00016=266052,556475
EC00017=371159,556475
EC00018=443420,556475
EC00019=443420,556475
EC00020=443420,556475
EC00021=443420,556475
EC00022=443420,556475
EC00023=443420,556475
EC00024=443419,556475
EC00025=443420,556475
EC00026=443420,556475
EC00027=443420,556475
EC00028=443420,556475
EC00029=443420,556475
EC00030=443420,556475
EC00031=443420,556475
EC00032=443420,556475
EC00033=443420,556475
EC00034=443420,556475
EC00035=443420,556475
EC00036=443420,556475
EC00037=443420,556475
EC00038=443420,556475
EC00039=443420,556475
EC00040=443420,556475
EC00041=443420,556475
EC00042=443420,556475
EC00043=443420,556475
EC00044=443420,556475
EC00045=443420,556475
EC00046=443420,556475
EC00047=443420,556475
EC00048=443420,556475
EC00049=443420,556475
EC00050=443420,556475
EC00051=443420,556475
EC00052=443420,556475
EC00053=443420,556475
EC00054=443420,556475
EC00055=443420,556475
EC00056=443420,556475
EC00057=443420,556475
EC00058=443420,556475
EC00059=443420,556475
EC00060=287458,556475
EC00061=266052,556475
EC00062=266052,556475
EC00063=266052,556475
EC00064=266052,556475
EC00065=266052,556475
EC00066=266052,556475
EC00067=266052,556475
EC00068=266052,556475
EC00069=266052,556475
EC00070=266052,556475
EC00071=266052,556475
EC00072=266052,556475
EC00073=266052,556475
EC00074=266052,556475
EC00075=266052,556475
EC00076=266052,556475
EC00077=266052,556475
EC00078=266052,556475
EC00079=266052,556475
EC00080=266052,556475
EC00081=266052,556475
EC00082=266052,556475
EC00083=266052,556475
EC00084=266052,556475
EC00085=266052,556475
EC00086=266052,556475
EC00087=266052,556475
EC00088=266052,556475
EC00089=266052,556475
EC00090=266052,556475
EC00091=344235,556475
EC00092=443420,556475
EC00093=443420,556475
EC00094=443420,556475
EC00095=443420,556475
EC00096=443420,556475
EC00097=443420,556475
EC00098=443420,556475
EC00099=443420,556475
EC00100=443420,556475
EC00101=443420,556475
EC00102=443420,556475
EC00103=443420,556475
EC00104=443420,556475
EC00105=443420,556475
EC00106=443420,556475
EC00107=443420,556475
EC00108=443420,556475
EC00109=443420,556475
EC00110=443420,556475
EC00111=443420,556475
EC00112=443420,556475
EC00113=443420,556475
EC00114=443420,556475
EC00115=443420,556475
EC00116=443420,556475
EC00117=443420,556475
EC00118=443420,556475
EC00119=443420,556475
EC00120=443420,556475
EC00121=443420,556475
EC00122=443420,556475
EC00123=443420,556475
EC00124=443420,556475
EC00125=443420,556475
EC00126=443420,556475
EC00127=443420,556475
EC00128=443420,556475
EC00129=443420,556475
EC00130=443420,556475
EC00131=443420,556475
EC00132=443420,556475
EC00133=443420,556475
EC00134=443420,556475
EC00135=443420,556475
EC00136=443420,556475
EC00137=492425,556475
EC00138=492425,556475
EC00139=492424,556474
EC00140=492424,556474
EC00141=492424,556474
EC00142=492424,556474
EC00143=492424,556474
EC00144=492424,556474
EC00145=492424,556474
EC00146=492424,556474
EC00147=492424,556474
EC00148=492424,556474
EC00149=492424,556474
EC00150=492425,556475
EC00151=492424,556474
EC00152=492424,556474
EC00153=492424,556474
EC00154=492424,556474
EC00155=492424,556474
EC00156=492424,556474
EC00157=492424,556474
EC00158=492424,556474
EC00159=492424,556474
EC00160=492424,556474
EC00161=492424,556474
EC00162=492425,556475
EC00163=492424,556474
EC00164=492424,556474
EC00165=492424,556474
EC00166=492424,556474
EC00167=492424,556474
EC00168=492424,556474
EC00169=492424,556474
EC00170=492424,556474
EC00171=492424,556474
EC00172=492424,556474
EC00173=492424,556474
EC00174=492424,556474
EC00175=492425,556475
EC00176=492424,556474
EC00177=492424,556474
EC00178=492424,556474
EC00179=492424,556474
EC00180=492424,556474
EC00181=492424,556474
EC00182=492424,556474
EC00183=492424,556474
EC00184=492424,556474
EC00185=492424,556474
EC00186=492424,556474
EC00187=492425,556475
EC00188=492424,556474
EC00189=492424,556474
EC00190=492424,556474
EC00191=492424,556474
EC00192=492424,556474
EC00193=492424,556474
EC00194=492424,556474
EC00195=492424,556474
EC00196=492424,556474
EC00197=492424,556474
EC00198=492424,556474
EC00199=492425,556475
EC00200=492424,556474
EC00201=492424,556474
EC00202=492424,556474
EC00203=492424,556474
EC00204=492424,556474
EC00205=492424,556474
EC00206=492424,556474
EC00207=492424,556474
EC00208=492424,556474
EC00209=492424,556474
EC00210=492424,556474
EC00211=492425,556475
EC00212=492424,556474
EC00213=492424,556474
EC00214=492424,556474
EC00215=492424,556474
EC00216=492424,556474
EC00217=492424,556474
EC00218=492424,556474
EC00219=492424,556474
EC00220=492424,556474
EC00221=492424,556474
EC00222=492424,556474
EC00223=492424,556474
EC00224=492424,556474
EC00225=492425,556475
EC00226=492424,556474
EC00227=492424,556474
EC00228=492424,556474
EC00229=492424,556474
EC00230=492424,556474
EC00231=492424,556474
EC00232=492424,556474
EC00233=492424,556474
EC00234=492424,556474
EC00235=492424,556474
EC00236=492424,556474
EC00237=492424,556474
EC00238=492425,556475
EC00239=492424,556474
EC00240=492424,556474
EC00241=492424,556474
EC00242=492424,556474
EC00243=492424,556474
EC00244=492424,556474
EC00245=492424,556474
EC00246=492424,556474
EC00247=492424,556474
EC00248=492424,556474
EC00249=492424,556474
EC00250=492424,556474
EC00251=492424,556474
EC00252=492425,556475
EC00253=492424,556474
EC00254=492424,556474
EC00255=492423,556474
EC00256=492424,556474
EC00257=492424,556474
EC00258=492424,556474
EC00259=492424,556474
EC00260=492424,556474
EC00261=492424,556474
EC00262=492424,556474
EC00263=492424,556474
EC00264=492424,556474
EC00265=492425,556475
EC00266=266052,556475
EC00267=266052,556475
EC00268=266052,556475
EC00269=266052,556475
EC00270=266052,556475
EC00271=266052,556475
EC00272=266052,556475
EC00273=266052,556475
EC00274=266052,556475
EC00275=266052,556475
EC00276=266052,556475
EC00277=266052,556475
EC00278=266052,556475
EC00279=266052,556475
EC00280=266052,556475
EC00281=266052,556475
EC00282=266052,556475
EC00283=266052,556475
EC00284=266052,556475
EC00285=266052,556475
EC00286=266052,556475
EC00287=266052,556475
EC00288=266052,556475
EC00289=266052,556475
EC00290=266052,556475
EC00291=266052,556475
EC00292=266052,556475
EC00293=266052,556475
EC00294=266052,556475
EC00295=266052,556475
EC00296=266052,556475
EC00297=266052,556475
EC00298=266052,556475
EC00299=266052,556475
EC00300=266052,556475
EC00301=266052,556475
EC00302=266052,556475
EC00303=266052,556475
EC00304=266052,556475
EC00305=266052,556475
EC00306=266052,556475
EC00307=266052,556475
EC00308=266052,556475
EC00309=266052,556475
EC00310=266052,556475
EC00311=266052,556475
EC00312=266052,556475
EC00313=266052,556475
EC00314=266052,556475
EC00315=266052,556475
EC00316=266052,556475
EC00317=266052,556475
EC00318=266052,556475
EC00319=266052,556475
EC00320=266052,556475
EC00321=266052,556475
EC00322=266052,556475
EC00323=266052,556475
EC00324=266052,556475
EC00325=266052,556475
EC00326=266052,556475
EC00327=266052,556475
EC00328=266052,556475
EC00329=266052,556475
EC00330=266052,556475
EC00331=266052,556475
EC00332=266052,556475
EC00333=266052,556475
EC00334=266052,556475
EC00335=266052,556475
EC00336=266052,556475
EC00337=266052,556475
EC00338=266052,556475
EC00339=266052,556475
EC00340=266052,556475
EC00341=266052,556475
EC00342=266052,556475
EC00343=266052,556475
EC00344=266052,556475
EC00345=266052,556475
EC00346=266052,556475
EC00347=266052,556475
EC00348=266052,556475
EC00349=266052,556475
EC00350=266052,556475
EC00351=266052,556475
EC00352=266052,556475
EC00353=266052,556475
EC00354=266052,556475
EC00355=266052,556475
EC00356=266052,556475
EC00357=266052,556475
EC00358=266052,556475
EC00359=266052,556475
EC00360=266052,556475
EC00361=266052,556475
EC00362=266052,556475
EC00363=266052,556475
EC00364=266052,556475
EC00365=266052,556475
EC00366=266052,556475
EC00367=266052,556475
EC00368=266052,556475
EC00369=266052,556475
EC00370=266052,556475
EC00371=266052,556475
EC00372=266052,556475
EC00373=266052,556475
EC00374=266052,556475
EC00375=266052,556475
EC00376=266052,556475
EC00377=266052,556475
EC00378=266052,556475
EC00379=266052,556475
EC00380=266052,556475
EC00381=266052,556475
EC00382=266052,556475
EC00383=266052,556475
EC00384=266052,556475
EC00385=266052,556475
EC00386=266052,556475
EC00387=266052,556475
EC00388=266052,556475
EC00389=266052,556475
EC00390=266052,556475
EC00391=266052,556475
EC00392=266052,556475
EC00393=266052,556475
EC00394=266052,556475
EC00395=266052,556475
EC00396=266052,556475
EC00397=266052,556475
EC00398=266052,556475
EC00399=266052,556475
EC00400=266052,556475
EC00401=266052,556475
EC00402=266052,556475
EC00403=266052,556475
EC00404=266052,556475
EC00405=266052,556475
EC00406=266052,556475
EC00407=266052,556475
EC00408=266052,556475
EC00409=266052,556475
EC00410=266052,556475
EC00411=266052,556475
EC00412=266052,556475
EC00413=266052,556475
EC00414=266052,556475
EC00415=266052,556475
EC00416=266052,556475
EC00417=266052,556475
EC00418=266052,556475
EC00419=266052,556475
EC00420=266052,556475
EC00421=266052,556475
EC00422=266052,556475
EC00423=266052,556475
EC00424=266052,556475
EC00425=266052,556475
EC00426=266052,556475
EC00427=266052,556475
EC00428=266052,556475
EC00429=266052,556475
EC00430=266052,556475
EC00431=266052,556475
EC00432=266052,556475
EC00433=266052,556475
EC00434=347188,556475
EC00435=443420,556475
EC00436=443420,556475
EC00437=443420,556475
EC00438=443420,556475
EC00439=443420,556475
EC00440=443420,556475
EC00441=443420,556475
EC00442=443420,556475
EC00443=443420,556475
EC00444=443420,556475
EC00445=443420,556475
EC00446=443420,556475
EC00447=443420,556475
EC00448=443420,556475
EC00449=443420,556475
EC00450=443420,556475
EC00451=443420,556475
EC00452=443420,556475
EC00453=443419,556475
EC00454=443419,556475
EC00455=443420,556475
EC00456=443420,556475
EC00457=443420,556475
EC00458=443420,556475
EC00459=443420,556475
EC00460=443420,556475
EC00461=443420,556475
EC00462=443420,556475
EC00463=443420,556475
EC00464=443420,556475
EC00465=443420,556475
EC00466=443420,556475
EC00467=443420,556475
EC00468=443420,556475
EC00469=443420,556475
EC00470=443420,556475
EC00471=443420,556475
EC00472=443420,556475
EC00473=443420,556475
EC00474=443420,556475
EC00475=443420,556475
EC00476=443420,556475
EC00477=443420,556475
EC00478=443420,556475
EC00479=443420,556475
EC00480=443420,556475
EC00481=443420,556475
EC00482=443420,556475
EC00483=443420,556475
EC00484=443420,556475
EC00485=443420,556475
EC00486=443420,556475
EC00487=443420,556475
EC00488=443420,556475
EC00489=443420,556475
EC00490=443420,556475
EC00491=443420,556475
EC00492=443420,556475
EC00493=443420,556475
EC00494=443420,556475
EC00495=443420,556475
EC00496=443420,556475
EC00497=443420,556475
EC00498=443420,556475
EC00499=443420,556475
EC00500=443420,556475
EC00501=443420,556475
EC00502=443420,556475
EC00503=443420,556475
EC00504=443420,556475
EC00505=443420,556475
EC00506=443420,556475
EC00507=443420,556475
EC00508=443420,556475
EC00509=443419,556475
EC00510=346238,556475
EC00511=305669,556475
EC00512=266052,556475
EC00513=266052,556475
EC00514=266052,556475
EC00515=266052,556475
EC00516=266052,556475
EC00517=266052,556475
EC00518=266052,556475
EC00519=266052,556475
EC00520=266052,556475
EC00521=266052,556475
EC00522=266052,556475
EC00523=266052,556475
EC00524=266052,556475
EC00525=266052,556475
EC00526=266052,556475
EC00527=266052,556475
EC00528=266052,556475
EC00529=266052,556475
EC00530=266052,556475
EC00531=266052,556475
EC00532=266052,556475
EC00533=266052,556475
EC00534=266052,556475
EC00535=266052,556475
EC00536=266052,556475
EC00537=266052,556475
EC00538=266052,556475
EC00539=266052,556475
EC00540=266052,556475
EC00541=266052,556475
EC00542=266052,556475
EC00543=266052,556475
EC00544=266052,556475
EC00545=266052,556475
EC00546=266052,556475
EC00547=266052,556475
EC00548=266052,556475
EC00549=266052,556475
EC00550=266052,556475
EC00551=266052,556475
EC00552=266052,556475
EC00553=266052,556475
EC00554=266052,556475
EC00555=266052,556475
EC00556=266052,556475
EC00557=266052,556475
EC00558=443420,556475
EC00559=443420,556475
///POSTYPE BASE
///RECTAN
///RCONF 0,0,0,0,0,0,0,0,0,0,0,0,0,0,0,0,0,0,0,0,0,0,0,0
P00006=0.222,-3.123,-1.508,0.0000,0.0000,0.0000
P00021=-0.225,-6.128,-0.405,0.0000,0.0000,0.0000
P00022=0.222,-3.123,-1.508,0.0000,0.0000,0.0000
P00031=1.853,-0.001,-1.549,0.0000,0.0000,0.0000
P00032=1.957,0.503,-7.217,0.0000,0.0000,0.0000
///RCONF 0,0,0,0,1,0,0,0,0,0,0,0,0,0,0,0,0,0,0,0,0,0,0,0
P00033=-0.123,0.612,-5.012,0.0000,0.0000,0.0000
///RCONF 0,0,0,0,0,0,0,0,0,0,0,0,0,0,0,0,0,0,0,0,0,0,0,0
P00034=-0.304,0.773,-2.693,0.0000,0.0000,0.0000
P00035=2.817,0.591,-1.622,0.0000,0.0000,0.0000
P00036=-1.108,-0.829,1.850,0.0000,0.0000,0.0000
P00040=-0.030,9.648,2.467,0.0000,0.0000,0.0000
P00041=0.192,3.924,0.305,0.0000,0.0000,0.0000
P00042=-0.217,1.941,0.413,0.0000,0.0000,0.0000
P00043=-0.044,-1.937,1.197,0.0000,0.0000,0.0000
P00044=0.687,-2.322,1.156,0.0000,0.0000,0.0000
P00045=-0.068,-0.810,1.603,0.0000,0.0000,0.0000
P00050=4.296,-4.501,-0.826,0.0000,0.0000,0.0000
P00051=0.367,3.892,0.009,0.0000,0.0000,0.0000
P00052=0.088,2.832,-0.342,0.0000,0.0000,0.0000
P00053=0.134,6.594,0.107,0.0000,0.0000,0.0000
P00054=-0.103,6.509,-0.702,0.0000,0.0000,0.0000
P00055=-0.342,8.912,1.324,0.0000,0.0000,0.0000
//INST
///DATE 2025/05/19 14:56
///ATTR SC,RW
///GROUP1 RB1,BS1
///GROUP2 ST1
NOP
'X2_103(30,90)
MOVJ C00000 BC00000 VJ=100.00  +MOVJ EC00000 VJ=100.00
MOVJ C00001 BC00001 VJ=100.00  +MOVJ EC00001 VJ=100.00
MOVJ C00002 BC00002 VJ=100.00  +MOVJ EC00002 VJ=100.00
MOVJ C00003 BC00003 VJ=15.00  +MOVJ EC00003 VJ=100.00
'Path S4757
SFTOF3D
COMM PAUSE
COMM MOVJ C00004 BC00004 VJ=100.00  +MOVJ EC00004 VJ=100.00
COMM MOVL C00005 BC00005 V=800.0  +MOVJ EC00005 VJ=100.00
COMM SMOVL C00006 BC00006 V=166.7  +MOVJ EC00006
COMM SMOVL C00007 BC00007 V=166.7  +MOVJ EC00007
COMM SREFP 3 C00008 BC00008  +REFP EC00008
COMM CALL JOB:SEARCH-R1-S13D
COMM SET P040 P006
COMM SFTON3D P040
COMM SMOVL C00009 BC00009 V=166.7  +MOVJ EC00009
COMM SMOVL C00010 BC00010 V=166.7  +MOVJ EC00010
COMM SMOVL C00011 BC00011 V=100.0  +MOVJ EC00011
COMM SREFP 3 C00012 BC00012  +REFP EC00012
COMM CALL JOB:SEARCH-R1-S13D
COMM SET P040 P006
COMM SFTON3D P040
COMM SMOVL C00013 BC00013 V=166.7  +MOVJ EC00013
COMM MOVL C00014 BC00014 V=800.0  +MOVJ EC00014 VJ=100.00
COMM MOVL C00015 BC00015 V=1000.0  +MOVJ EC00015 VJ=100.00
'EndPath S4757
MOVJ C00016 BC00016 VJ=100.00  +MOVJ EC00016 VJ=100.00
MOVJ C00017 BC00017 VJ=100.00  +MOVJ EC00017 VJ=100.00
'Path S4795
SFTOF3D
MOVJ C00018 BC00018 VJ=100.00  +MOVJ EC00018 VJ=100.00
MOVL C00019 BC00019 V=800.0  +MOVJ EC00019 VJ=100.00
SMOVL C00020 BC00020 V=166.7  +MOVJ EC00020
SREFP 3 C00021 BC00021  +REFP EC00021
CALL JOB:SEARCH-R1-S13D
SET P031 P006
SFTON3D P031
SMOVL C00022 BC00022 V=166.7  +MOVJ EC00022
SMOVL C00023 BC00023 V=166.7  +MOVJ EC00023
SREFP 3 C00024 BC00024  +REFP EC00024
CALL JOB:SEARCH-R1-S13D
SET P031 P006
SFTON3D P031
SMOVL C00025 BC00025 V=166.7  +MOVJ EC00025
SMOVL C00026 BC00026 V=166.7  +MOVJ EC00026
SREFP 3 C00027 BC00027  +REFP EC00027
CALL JOB:SEARCH-R1-S13D
SET P031 P006
SFTON3D P031
SMOVL C00028 BC00028 V=166.7  +MOVJ EC00028
MOVL C00029 BC00029 V=800.0  +MOVJ EC00029 VJ=100.00
MOVL C00030 BC00030 V=1000.0  +MOVJ EC00030 VJ=100.00
'EndPath S4795
MOVJ C00031 BC00031 VJ=100.00  +MOVJ EC00031 VJ=100.00
'Path S4863
SFTOF3D
MOVJ C00032 BC00032 VJ=100.00  +MOVJ EC00032 VJ=100.00
MOVL C00033 BC00033 V=800.0  +MOVJ EC00033 VJ=100.00
SMOVL C00034 BC00034 V=166.7  +MOVJ EC00034
SREFP 3 C00035 BC00035  +REFP EC00035
CALL JOB:SEARCH-R1-S13D
SET P032 P006
SFTON3D P032
SMOVL C00036 BC00036 V=166.7  +MOVJ EC00036
SMOVL C00037 BC00037 V=166.7  +MOVJ EC00037
SREFP 3 C00038 BC00038  +REFP EC00038
CALL JOB:SEARCH-R1-S13D
SET P032 P006
SFTON3D P032
SMOVL C00039 BC00039 V=166.7  +MOVJ EC00039
SMOVL C00040 BC00040 V=166.7  +MOVJ EC00040
SREFP 3 C00041 BC00041  +REFP EC00041
CALL JOB:SEARCH-R1-S13D
SET P032 P006
SFTON3D P032
SMOVL C00042 BC00042 V=166.7  +MOVJ EC00042
MOVL C00043 BC00043 V=800.0  +MOVJ EC00043 VJ=100.00
MOVL C00044 BC00044 V=1000.0  +MOVJ EC00044 VJ=100.00
'EndPath S4863
MOVJ C00045 BC00045 VJ=100.00  +MOVJ EC00045 VJ=100.00
'Path S4864
SFTOF3D
MOVJ C00046 BC00046 VJ=100.00  +MOVJ EC00046 VJ=100.00
MOVL C00047 BC00047 V=800.0  +MOVJ EC00047 VJ=100.00
SMOVL C00048 BC00048 V=166.7  +MOVJ EC00048
SREFP 3 C00049 BC00049  +REFP EC00049
CALL JOB:SEARCH-R1-S13D
SET P033 P006
SFTON3D P033
SMOVL C00050 BC00050 V=166.7  +MOVJ EC00050
SMOVL C00051 BC00051 V=166.7  +MOVJ EC00051
SREFP 3 C00052 BC00052  +REFP EC00052
CALL JOB:SEARCH-R1-S13D
SET P033 P006
SFTON3D P033
SMOVL C00053 BC00053 V=166.7  +MOVJ EC00053
SMOVL C00054 BC00054 V=333.3  +MOVJ EC00054
SMOVL C00055 BC00055 V=166.7  +MOVJ EC00055
SREFP 3 C00056 BC00056  +REFP EC00056
CALL JOB:SEARCH-R1-S13D
SET P033 P006
SFTON3D P033
SMOVL C00057 BC00057 V=166.7  +MOVJ EC00057
SMOVL C00058 BC00058 V=166.7  +MOVJ EC00058
MOVL C00059 BC00059 V=1000.0  +MOVJ EC00059 VJ=100.00
'EndPath S4864
MOVJ C00060 BC00060 VJ=100.00  +MOVJ EC00060 VJ=100.00
'Path S4786
SFTOF3D
MOVJ C00061 BC00061 VJ=100.00  +MOVJ EC00061 VJ=100.00
MOVL C00062 BC00062 V=800.0  +MOVJ EC00062 VJ=100.00
SMOVL C00063 BC00063 V=166.7  +MOVJ EC00063
SREFP 3 C00064 BC00064  +REFP EC00064
CALL JOB:SEARCH-R1-S13D
SET P021 P006
SFTON3D P021
SMOVL C00065 BC00065 V=166.7  +MOVJ EC00065
SMOVL C00066 BC00066 V=166.7  +MOVJ EC00066
SREFP 3 C00067 BC00067  +REFP EC00067
CALL JOB:SEARCH-R1-S13D
SET P021 P006
SFTON3D P021
SMOVL C00068 BC00068 V=166.7  +MOVJ EC00068
SMOVL C00069 BC00069 V=166.7  +MOVJ EC00069
SREFP 3 C00070 BC00070  +REFP EC00070
CALL JOB:SEARCH-R1-S13D
SET P021 P006
SFTON3D P021
SMOVL C00071 BC00071 V=166.7  +MOVJ EC00071
MOVL C00072 BC00072 V=800.0  +MOVJ EC00072 VJ=100.00
MOVL C00073 BC00073 V=1000.0  +MOVJ EC00073 VJ=100.00
'EndPath S4786
MOVJ C00074 BC00074 VJ=100.00  +MOVJ EC00074 VJ=100.00
MOVJ C00075 BC00075 VJ=100.00  +MOVJ EC00075 VJ=100.00
MOVJ C00076 BC00076 VJ=100.00  +MOVJ EC00076 VJ=100.00
'Path S4787
SFTOF3D
MOVJ C00077 BC00077 VJ=100.00  +MOVJ EC00077 VJ=100.00
MOVL C00078 BC00078 V=800.0  +MOVJ EC00078 VJ=100.00
SMOVL C00079 BC00079 V=166.7  +MOVJ EC00079
SREFP 3 C00080 BC00080  +REFP EC00080
CALL JOB:SEARCH-R1-S13D
SET P022 P006
SFTON3D P022
SMOVL C00081 BC00081 V=166.7  +MOVJ EC00081
SMOVL C00082 BC00082 V=166.7  +MOVJ EC00082
SREFP 3 C00083 BC00083  +REFP EC00083
CALL JOB:SEARCH-R1-S13D
SET P022 P006
SFTON3D P022
SMOVL C00084 BC00084 V=166.7  +MOVJ EC00084
SMOVL C00085 BC00085 V=166.7  +MOVJ EC00085
SREFP 3 C00086 BC00086  +REFP EC00086
CALL JOB:SEARCH-R1-S13D
SET P022 P006
SFTON3D P022
SMOVL C00087 BC00087 V=166.7  +MOVJ EC00087
MOVL C00088 BC00088 V=800.0  +MOVJ EC00088 VJ=100.00
MOVL C00089 BC00089 V=1000.0  +MOVJ EC00089 VJ=100.00
'EndPath S4787
MOVJ C00090 BC00090 VJ=100.00  +MOVJ EC00090 VJ=100.00
MOVJ C00091 BC00091 VJ=100.00  +MOVJ EC00091 VJ=100.00
'Path S4800
SFTOF3D
MOVJ C00092 BC00092 VJ=100.00  +MOVJ EC00092 VJ=100.00
MOVL C00093 BC00093 V=800.0  +MOVJ EC00093 VJ=100.00
SMOVL C00094 BC00094 V=166.7  +MOVJ EC00094
SREFP 3 C00095 BC00095  +REFP EC00095
CALL JOB:SEARCH-R1-S13D
SET P036 P006
SFTON3D P036
SMOVL C00096 BC00096 V=166.7  +MOVJ EC00096
SMOVL C00097 BC00097 V=166.7  +MOVJ EC00097
SREFP 3 C00098 BC00098  +REFP EC00098
CALL JOB:SEARCH-R1-S13D
SET P036 P006
SFTON3D P036
SMOVL C00099 BC00099 V=166.7  +MOVJ EC00099
SMOVL C00100 BC00100 V=166.7  +MOVJ EC00100
SMOVL C00101 BC00101 V=166.7  +MOVJ EC00101
SREFP 3 C00102 BC00102  +REFP EC00102
CALL JOB:SEARCH-R1-S13D
SET P036 P006
SFTON3D P036
SMOVL C00103 BC00103 V=166.7  +MOVJ EC00103
SMOVL C00104 BC00104 V=166.7  +MOVJ EC00104
SMOVL C00105 BC00105 V=166.7  +MOVJ EC00105
MOVL C00106 BC00106 V=800.0  +MOVJ EC00106 VJ=100.00
MOVL C00107 BC00107 V=1000.0  +MOVJ EC00107 VJ=100.00
'EndPath S4800
MOVJ C00108 BC00108 VJ=100.00  +MOVJ EC00108 VJ=100.00
'Path S4799
SFTOF3D
MOVJ C00109 BC00109 VJ=100.00  +MOVJ EC00109 VJ=100.00
MOVL C00110 BC00110 V=800.0  +MOVJ EC00110 VJ=100.00
SMOVL C00111 BC00111 V=166.7  +MOVJ EC00111
SREFP 3 C00112 BC00112  +REFP EC00112
CALL JOB:SEARCH-R1-S13D
SET P035 P006
SFTON3D P035
SMOVL C00113 BC00113 V=166.7  +MOVJ EC00113
SMOVL C00114 BC00114 V=166.7  +MOVJ EC00114
SREFP 3 C00115 BC00115  +REFP EC00115
CALL JOB:SEARCH-R1-S13D
SET P035 P006
SFTON3D P035
SMOVL C00116 BC00116 V=166.7  +MOVJ EC00116
SMOVL C00117 BC00117 V=166.7  +MOVJ EC00117
SREFP 3 C00118 BC00118  +REFP EC00118
CALL JOB:SEARCH-R1-S13D
SET P035 P006
SFTON3D P035
SMOVL C00119 BC00119 V=166.7  +MOVJ EC00119
MOVL C00120 BC00120 V=800.0  +MOVJ EC00120 VJ=100.00
MOVL C00121 BC00121 V=1000.0  +MOVJ EC00121 VJ=100.00
'EndPath S4799
MOVJ C00122 BC00122 VJ=100.00  +MOVJ EC00122 VJ=100.00
'Path S4798
SFTOF3D
MOVJ C00123 BC00123 VJ=100.00  +MOVJ EC00123 VJ=100.00
MOVL C00124 BC00124 V=800.0  +MOVJ EC00124 VJ=100.00
SMOVL C00125 BC00125 V=166.7  +MOVJ EC00125
SREFP 3 C00126 BC00126  +REFP EC00126
CALL JOB:SEARCH-R1-S13D
SET P034 P006
SFTON3D P034
SMOVL C00127 BC00127 V=166.7  +MOVJ EC00127
SMOVL C00128 BC00128 V=166.7  +MOVJ EC00128
SREFP 3 C00129 BC00129  +REFP EC00129
CALL JOB:SEARCH-R1-S13D
SET P034 P006
SFTON3D P034
SMOVL C00130 BC00130 V=166.7  +MOVJ EC00130
SMOVL C00131 BC00131 V=166.7  +MOVJ EC00131
SREFP 3 C00132 BC00132  +REFP EC00132
CALL JOB:SEARCH-R1-S13D
SET P034 P006
SFTON3D P034
SMOVL C00133 BC00133 V=166.7  +MOVJ EC00133
MOVL C00134 BC00134 V=800.0  +MOVJ EC00134 VJ=100.00
MOVL C00135 BC00135 V=1000.0  +MOVJ EC00135 VJ=100.00
'EndPath S4798
MOVJ C00136 BC00136 VJ=100.00  +MOVJ EC00136 VJ=100.00
MOVJ C00137 BC00137 VJ=100.00  +MOVJ EC00137 VJ=100.00
'Path S4780
SFTOF3D
MOVL C00138 BC00138 V=666.7  +MOVJ EC00138 VJ=100.00
SMOVL C00139 BC00139 V=166.7  +MOVJ EC00139
SREFP 3 C00140 BC00140  +REFP EC00140
CALL JOB:SEARCH-R1-S13D
SET P041 P006
SFTON3D P041
SMOVL C00141 BC00141 V=166.7  +MOVJ EC00141
SREFP 3 C00142 BC00142  +REFP EC00142
CALL JOB:SEARCH-R1-S13D
SET P041 P006
SFTON3D P041
SMOVL C00143 BC00143 V=166.7  +MOVJ EC00143
SMOVL C00144 BC00144 V=166.7  +MOVJ EC00144
SMOVL C00145 BC00145 V=166.7  +MOVJ EC00145
SREFP 3 C00146 BC00146  +REFP EC00146
CALL JOB:SEARCH-R1-S13D
SET P051 P006
SFTON3D P051
SMOVL C00147 BC00147 V=100.0  +MOVJ EC00147
SREFP 3 C00148 BC00148  +REFP EC00148
CALL JOB:SEARCH-R1-S13D
SET P051 P006
SFTON3D P051
SMOVL C00149 BC00149 V=166.7  +MOVJ EC00149
SFTOF3D
MOVL C00150 BC00150 V=666.7  +MOVJ EC00150 VJ=100.00
SMOVL C00151 BC00151 V=166.7  +MOVJ EC00151
SREFP 3 C00152 BC00152  +REFP EC00152
CALL JOB:SEARCH-R1-S13D
SET P042 P006
SFTON3D P042
SMOVL C00153 BC00153 V=166.7  +MOVJ EC00153
SREFP 3 C00154 BC00154  +REFP EC00154
CALL JOB:SEARCH-R1-S13D
SET P042 P006
SFTON3D P042
SMOVL C00155 BC00155 V=166.7  +MOVJ EC00155
SMOVL C00156 BC00156 V=166.7  +MOVJ EC00156
SMOVL C00157 BC00157 V=166.7  +MOVJ EC00157
SREFP 3 C00158 BC00158  +REFP EC00158
CALL JOB:SEARCH-R1-S13D
SET P052 P006
SFTON3D P052
SMOVL C00159 BC00159 V=100.0  +MOVJ EC00159
SREFP 3 C00160 BC00160  +REFP EC00160
CALL JOB:SEARCH-R1-S13D
SET P052 P006
SFTON3D P052
SMOVL C00161 BC00161 V=166.7  +MOVJ EC00161
SFTOF3D
MOVL C00162 BC00162 V=666.7  +MOVJ EC00162 VJ=100.00
SMOVL C00163 BC00163 V=166.7  +MOVJ EC00163
SREFP 3 C00164 BC00164  +REFP EC00164
CALL JOB:SEARCH-R1-S13D
SET P043 P006
SFTON3D P043
SMOVL C00165 BC00165 V=166.7  +MOVJ EC00165
SREFP 3 C00166 BC00166  +REFP EC00166
CALL JOB:SEARCH-R1-S13D
SET P043 P006
SFTON3D P043
SMOVL C00167 BC00167 V=166.7  +MOVJ EC00167
SMOVL C00168 BC00168 V=166.7  +MOVJ EC00168
SMOVL C00169 BC00169 V=166.7  +MOVJ EC00169
SREFP 3 C00170 BC00170  +REFP EC00170
CALL JOB:SEARCH-R1-S13D
SET P053 P006
SFTON3D P053
SMOVL C00171 BC00171 V=100.0  +MOVJ EC00171
SREFP 3 C00172 BC00172  +REFP EC00172
CALL JOB:SEARCH-R1-S13D
SET P053 P006
SFTON3D P053
SMOVL C00173 BC00173 V=166.7  +MOVJ EC00173
SFTOF3D
MOVL C00174 BC00174 V=666.7  +MOVJ EC00174 VJ=100.00
MOVL C00175 BC00175 V=666.7  +MOVJ EC00175 VJ=100.00
SMOVL C00176 BC00176 V=166.7  +MOVJ EC00176
SREFP 3 C00177 BC00177  +REFP EC00177
CALL JOB:SEARCH-R1-S13D
SET P044 P006
SFTON3D P044
SMOVL C00178 BC00178 V=166.7  +MOVJ EC00178
SREFP 3 C00179 BC00179  +REFP EC00179
CALL JOB:SEARCH-R1-S13D
SET P044 P006
SFTON3D P044
SMOVL C00180 BC00180 V=166.7  +MOVJ EC00180
SMOVL C00181 BC00181 V=166.7  +MOVJ EC00181
SMOVL C00182 BC00182 V=166.7  +MOVJ EC00182
SREFP 3 C00183 BC00183  +REFP EC00183
CALL JOB:SEARCH-R1-S13D
SET P054 P006
SFTON3D P054
SMOVL C00184 BC00184 V=100.0  +MOVJ EC00184
SREFP 3 C00185 BC00185  +REFP EC00185
CALL JOB:SEARCH-R1-S13D
SET P054 P006
SFTON3D P054
SMOVL C00186 BC00186 V=166.7  +MOVJ EC00186
SFTOF3D
MOVL C00187 BC00187 V=666.7  +MOVJ EC00187 VJ=100.00
SMOVL C00188 BC00188 V=166.7  +MOVJ EC00188
SREFP 3 C00189 BC00189  +REFP EC00189
CALL JOB:SEARCH-R1-S13D
SET P045 P006
SFTON3D P045
SMOVL C00190 BC00190 V=166.7  +MOVJ EC00190
SREFP 3 C00191 BC00191  +REFP EC00191
CALL JOB:SEARCH-R1-S13D
SET P045 P006
SFTON3D P045
SMOVL C00192 BC00192 V=166.7  +MOVJ EC00192
SMOVL C00193 BC00193 V=166.7  +MOVJ EC00193
SMOVL C00194 BC00194 V=166.7  +MOVJ EC00194
SREFP 3 C00195 BC00195  +REFP EC00195
CALL JOB:SEARCH-R1-S13D
SET P055 P006
SFTON3D P055
SMOVL C00196 BC00196 V=100.0  +MOVJ EC00196
SREFP 3 C00197 BC00197  +REFP EC00197
CALL JOB:SEARCH-R1-S13D
SET P055 P006
SFTON3D P055
SMOVL C00198 BC00198 V=166.7  +MOVJ EC00198
SFTOF3D
MOVL C00199 BC00199 V=666.7  +MOVJ EC00199 VJ=100.00
SMOVL C00200 BC00200 V=166.7  +MOVJ EC00200
SREFP 3 C00201 BC00201  +REFP EC00201
CALL JOB:SEARCH-R1-S13D
SET P040 P006
SFTON3D P040
SMOVL C00202 BC00202 V=166.7  +MOVJ EC00202
SREFP 3 C00203 BC00203  +REFP EC00203
CALL JOB:SEARCH-R1-S13D
SET P040 P006
SFTON3D P040
SMOVL C00204 BC00204 V=166.7  +MOVJ EC00204
SMOVL C00205 BC00205 V=166.7  +MOVJ EC00205
SMOVL C00206 BC00206 V=166.7  +MOVJ EC00206
SREFP 3 C00207 BC00207  +REFP EC00207
CALL JOB:SEARCH-R1-S13D
SET P050 P006
SFTON3D P050
SMOVL C00208 BC00208 V=100.0  +MOVJ EC00208
SREFP 3 C00209 BC00209  +REFP EC00209
CALL JOB:SEARCH-R1-S13D
SET P050 P006
SFTON3D P050
SMOVL C00210 BC00210 V=166.7  +MOVJ EC00210
SFTOF3D
MOVL C00211 BC00211 V=666.7  +MOVJ EC00211 VJ=100.00
SFTON3D P044
SMOVL C00212 BC00212 V=166.7  +MOVJ EC00212
SMOVL C00213 BC00213 V=166.7 PL=0  +MOVJ EC00213
MACRO1 MJ#(0) ARGF9
ARCON
SFTON3D P045
SMOVL C00214 BC00214 V=10.0  +MOVJ EC00214
ARCOF
MOVL C00215 BC00215 V=166.7  +MOVJ EC00215 VJ=100.00
SFTOF3D
SMOVL C00216 BC00216 V=666.7  +MOVJ EC00216
SMOVL C00217 BC00217 V=666.7  +MOVJ EC00217
MOVL C00218 BC00218 V=666.7  +MOVJ EC00218 VJ=100.00
SFTON3D P044
SMOVL C00219 BC00219 V=166.7  +MOVJ EC00219
SMOVL C00220 BC00220 V=166.7 PL=0  +MOVJ EC00220
MACRO1 MJ#(0) ARGF9
ARCON
SFTON3D P043
SMOVL C00221 BC00221 V=10.0  +MOVJ EC00221
SFTON3D P042
SMOVL C00222 BC00222 V=10.0  +MOVJ EC00222
ARCOF
MOVL C00223 BC00223 V=166.7  +MOVJ EC00223 VJ=100.00
SFTOF3D
SMOVL C00224 BC00224 V=666.7  +MOVJ EC00224
SFTOF3D
MOVL C00225 BC00225 V=666.7  +MOVJ EC00225 VJ=100.00
SFTON3D P045
SMOVL C00226 BC00226 V=166.7  +MOVJ EC00226
SMOVL C00227 BC00227 V=166.7 PL=0  +MOVJ EC00227
MACRO1 MJ#(0) ARGF9
ARCON
SFTON3D P040
SMOVL C00228 BC00228 V=10.0  +MOVJ EC00228
ARCOF
MOVL C00229 BC00229 V=166.7  +MOVJ EC00229 VJ=100.00
SFTOF3D
SMOVL C00230 BC00230 V=666.7  +MOVJ EC00230
SMOVL C00231 BC00231 V=666.7  +MOVJ EC00231
MOVL C00232 BC00232 V=666.7  +MOVJ EC00232 VJ=100.00
SFTON3D P042
SMOVL C00233 BC00233 V=166.7  +MOVJ EC00233
SMOVL C00234 BC00234 V=166.7 PL=0  +MOVJ EC00234
MACRO1 MJ#(0) ARGF9
ARCON
SFTON3D P041
SMOVL C00235 BC00235 V=10.0  +MOVJ EC00235
ARCOF
MOVL C00236 BC00236 V=166.7  +MOVJ EC00236 VJ=100.00
SFTOF3D
SMOVL C00237 BC00237 V=666.7  +MOVJ EC00237
MOVL C00238 BC00238 V=666.7  +MOVJ EC00238 VJ=100.00
SFTON3D P054
SMOVL C00239 BC00239 V=166.7  +MOVJ EC00239
SMOVL C00240 BC00240 V=166.7 PL=0  +MOVJ EC00240
MACRO1 MJ#(0) ARGF9
ARCON
SFTON3D P055
SMOVL C00241 BC00241 V=10.0  +MOVJ EC00241
ARCOF
MOVL C00242 BC00242 V=166.7  +MOVJ EC00242 VJ=100.00
SFTOF3D
SMOVL C00243 BC00243 V=666.7  +MOVJ EC00243
SMOVL C00244 BC00244 V=666.7  +MOVJ EC00244
MOVL C00245 BC00245 V=666.7  +MOVJ EC00245 VJ=100.00
SFTON3D P054
SMOVL C00246 BC00246 V=166.7  +MOVJ EC00246
SMOVL C00247 BC00247 V=166.7 PL=0  +MOVJ EC00247
MACRO1 MJ#(0) ARGF9
ARCON
SFTON3D P053
SMOVL C00248 BC00248 V=10.0  +MOVJ EC00248
SFTON3D P052
SMOVL C00249 BC00249 V=10.0  +MOVJ EC00249
ARCOF
MOVL C00250 BC00250 V=166.7  +MOVJ EC00250 VJ=100.00
SFTOF3D
SMOVL C00251 BC00251 V=666.7  +MOVJ EC00251
SFTOF3D
MOVL C00252 BC00252 V=666.7  +MOVJ EC00252 VJ=100.00
SFTON3D P055
SMOVL C00253 BC00253 V=166.7  +MOVJ EC00253
SMOVL C00254 BC00254 V=166.7 PL=0  +MOVJ EC00254
MACRO1 MJ#(0) ARGF9
ARCON
SFTON3D P050
SMOVL C00255 BC00255 V=10.0  +MOVJ EC00255
ARCOF
MOVL C00256 BC00256 V=166.7  +MOVJ EC00256 VJ=100.00
SFTOF3D
SMOVL C00257 BC00257 V=666.7  +MOVJ EC00257
SMOVL C00258 BC00258 V=666.7  +MOVJ EC00258
MOVL C00259 BC00259 V=666.7  +MOVJ EC00259 VJ=100.00
SFTON3D P052
SMOVL C00260 BC00260 V=166.7  +MOVJ EC00260
SMOVL C00261 BC00261 V=166.7 PL=0  +MOVJ EC00261
MACRO1 MJ#(0) ARGF9
ARCON
SFTON3D P051
SMOVL C00262 BC00262 V=10.0  +MOVJ EC00262
ARCOF
MOVL C00263 BC00263 V=166.7  +MOVJ EC00263 VJ=100.00
SFTOF3D
SMOVL C00264 BC00264 V=666.7  +MOVJ EC00264
COMM SFTOF3D
COMM MOVL C00265 BC00265 V=800.0  +MOVJ EC00265 VJ=100.00
COMM SMOVL C00266 BC00266 V=166.7  +MOVJ EC00266
COMM SMOVL C00267 BC00267 V=166.7  +MOVJ EC00267
COMM SREFP 3 C00268 BC00268  +REFP EC00268
COMM CALL JOB:SEARCH-R1-S13D
COMM SET P041 P006
COMM SFTON3D P041
COMM SMOVL C00269 BC00269 V=166.7  +MOVJ EC00269
COMM SMOVL C00270 BC00270 V=166.7  +MOVJ EC00270
COMM SMOVL C00271 BC00271 V=100.0  +MOVJ EC00271
COMM SREFP 3 C00272 BC00272  +REFP EC00272
COMM CALL JOB:SEARCH-R1-S13D
COMM SET P041 P006
COMM SFTON3D P041
COMM SMOVL C00273 BC00273 V=166.7  +MOVJ EC00273
COMM SMOVL C00274 BC00274 V=250.0  +MOVJ EC00274
COMM MOVL C00275 BC00275 V=1000.0  +MOVJ EC00275 VJ=100.00
COMM 'EndPath S4780
COMM 'Path W4762
COMM SFTOF3D
COMM SFTON3D P041
COMM MOVJ C00276 BC00276 VJ=100.00  +MOVJ EC00276 VJ=100.00
COMM SMOVL C00277 BC00277 V=800.0  +MOVJ EC00277
COMM SMOVL C00278 BC00278 V=150.0 PL=0  +MOVJ EC00278
COMM MACRO1 MJ#(0) ARGF9
COMM ARCON
COMM SMOVL C00279 BC00279 V=10.0  +MOVJ EC00279
COMM SMOVL C00280 BC00280 V=10.0  +MOVJ EC00280
COMM ARCOF
COMM SMOVL C00281 BC00281 V=800.0  +MOVJ EC00281
COMM SMOVL C00282 BC00282 V=1000.0  +MOVJ EC00282
COMM SFTOF3D
COMM 'EndPath W4762
COMM 'Path W4764
COMM SFTOF3D
COMM SFTON3D P041
COMM MOVJ C00283 BC00283 VJ=100.00  +MOVJ EC00283 VJ=100.00
COMM SMOVL C00284 BC00284 V=800.0  +MOVJ EC00284
COMM SMOVL C00285 BC00285 V=150.0 PL=0  +MOVJ EC00285
COMM ARCON
COMM SMOVL C00286 BC00286 V=10.0  +MOVJ EC00286
COMM SMOVL C00287 BC00287 V=10.0  +MOVJ EC00287
COMM ARCOF
COMM SMOVL C00288 BC00288 V=800.0  +MOVJ EC00288
COMM SMOVL C00289 BC00289 V=1000.0  +MOVJ EC00289
COMM SFTOF3D
COMM 'EndPath W4764
COMM 'Path W4766
COMM SFTOF3D
COMM SFTON3D P041
COMM MOVJ C00290 BC00290 VJ=100.00  +MOVJ EC00290 VJ=100.00
COMM SMOVL C00291 BC00291 V=800.0  +MOVJ EC00291
COMM SMOVL C00292 BC00292 V=150.0 PL=0  +MOVJ EC00292
COMM ARCON
COMM SMOVL C00293 BC00293 V=10.0  +MOVJ EC00293
COMM SMOVL C00294 BC00294 V=10.0  +MOVJ EC00294
COMM ARCOF
COMM SMOVL C00295 BC00295 V=800.0  +MOVJ EC00295
COMM SMOVL C00296 BC00296 V=1000.0  +MOVJ EC00296
COMM SFTOF3D
COMM 'EndPath W4766
COMM '
COMM MOVJ C00297 BC00297 VJ=100.00  +MOVJ EC00297 VJ=100.00
COMM 'Path W4767
COMM SFTOF3D
COMM SFTON3D P040
COMM MOVJ C00298 BC00298 VJ=100.00  +MOVJ EC00298 VJ=100.00
COMM SMOVL C00299 BC00299 V=800.0  +MOVJ EC00299
COMM SMOVL C00300 BC00300 V=150.0 PL=0  +MOVJ EC00300
COMM ARCON
COMM SMOVL C00301 BC00301 V=10.0  +MOVJ EC00301
COMM SMOVL C00302 BC00302 V=10.0  +MOVJ EC00302
COMM ARCOF
COMM SMOVL C00303 BC00303 V=800.0  +MOVJ EC00303
COMM SMOVL C00304 BC00304 V=1000.0  +MOVJ EC00304
COMM SFTOF3D
COMM 'EndPath W4767
COMM 'Path W4768
COMM SFTOF3D
COMM SFTON3D P040
COMM MOVJ C00305 BC00305 VJ=100.00  +MOVJ EC00305 VJ=100.00
COMM SMOVL C00306 BC00306 V=800.0  +MOVJ EC00306
COMM SMOVL C00307 BC00307 V=150.0 PL=0  +MOVJ EC00307
COMM ARCON
COMM SMOVL C00308 BC00308 V=10.0  +MOVJ EC00308
COMM SMOVL C00309 BC00309 V=10.0  +MOVJ EC00309
COMM ARCOF
COMM SMOVL C00310 BC00310 V=800.0  +MOVJ EC00310
COMM SMOVL C00311 BC00311 V=1000.0  +MOVJ EC00311
COMM SFTOF3D
COMM 'EndPath W4768
COMM 'Path W4769
COMM SFTOF3D
COMM SFTON3D P040
COMM MOVJ C00312 BC00312 VJ=100.00  +MOVJ EC00312 VJ=100.00
COMM SMOVL C00313 BC00313 V=800.0  +MOVJ EC00313
COMM SMOVL C00314 BC00314 V=150.0 PL=0  +MOVJ EC00314
COMM ARCON
COMM SMOVL C00315 BC00315 V=10.0  +MOVJ EC00315
COMM SMOVL C00316 BC00316 V=10.0  +MOVJ EC00316
COMM ARCOF
COMM SMOVL C00317 BC00317 V=800.0  +MOVJ EC00317
COMM SFTOF3D
COMM 'EndPath W4769
COMM '
COMM MOVJ C00318 BC00318 VJ=100.00  +MOVJ EC00318 VJ=100.00
COMM MOVJ C00319 BC00319 VJ=100.00  +MOVJ EC00319 VJ=100.00
COMM 'Path W4765
COMM SFTOF3D
COMM SFTON3D P041
COMM MOVJ C00320 BC00320 VJ=100.00  +MOVJ EC00320 VJ=100.00
COMM SMOVL C00321 BC00321 V=800.0  +MOVJ EC00321
COMM SMOVL C00322 BC00322 V=150.0 PL=0  +MOVJ EC00322
COMM ARCON
COMM SMOVL C00323 BC00323 V=10.0  +MOVJ EC00323
COMM ARCOF
COMM SMOVL C00324 BC00324 V=800.0  +MOVJ EC00324
COMM SMOVL C00325 BC00325 V=1000.0  +MOVJ EC00325
COMM SFTOF3D
COMM 'EndPath W4765
COMM MOVJ C00326 BC00326 VJ=100.00  +MOVJ EC00326 VJ=100.00
COMM 'Path W4770
COMM SFTOF3D
COMM SFTON3D P040
COMM MOVJ C00327 BC00327 VJ=100.00  +MOVJ EC00327 VJ=100.00
COMM SMOVL C00328 BC00328 V=800.0  +MOVJ EC00328
COMM SMOVL C00329 BC00329 V=150.0 PL=0  +MOVJ EC00329
COMM ARCON
COMM SMOVL C00330 BC00330 V=10.0  +MOVJ EC00330
COMM ARCOF
COMM SMOVL C00331 BC00331 V=800.0  +MOVJ EC00331
COMM SMOVL C00332 BC00332 V=1000.0  +MOVJ EC00332
COMM SFTOF3D
COMM 'EndPath W4770
COMM MOVJ C00333 BC00333 VJ=100.00  +MOVJ EC00333 VJ=100.00
COMM 'up
COMM MOVJ C00334 BC00334 VJ=100.00  +MOVJ EC00334 VJ=100.00
COMM 'Path W4774
COMM SFTOF3D
COMM SFTON3D P041
COMM MOVJ C00335 BC00335 VJ=100.00  +MOVJ EC00335 VJ=100.00
COMM SMOVL C00336 BC00336 V=800.0  +MOVJ EC00336
COMM SMOVL C00337 BC00337 V=150.0 PL=0  +MOVJ EC00337
COMM MACRO1 MJ#(0) ARGF14
COMM ARCON
COMM SMOVL C00338 BC00338 V=10.0  +MOVJ EC00338
COMM SMOVL C00339 BC00339 V=10.0  +MOVJ EC00339
COMM ARCOF
COMM SMOVL C00340 BC00340 V=800.0  +MOVJ EC00340
COMM SMOVL C00341 BC00341 V=1000.0  +MOVJ EC00341
COMM SFTOF3D
COMM 'EndPath W4774
COMM 'Path W4788
COMM SFTOF3D
COMM SFTON3D P041
COMM MOVJ C00342 BC00342 VJ=100.00  +MOVJ EC00342 VJ=100.00
COMM SMOVL C00343 BC00343 V=800.0  +MOVJ EC00343
COMM SMOVL C00344 BC00344 V=150.0 PL=0  +MOVJ EC00344
COMM MACRO1 MJ#(0) ARGF9
COMM ARCON
COMM SMOVL C00345 BC00345 V=10.0  +MOVJ EC00345
COMM SMOVL C00346 BC00346 V=10.0  +MOVJ EC00346
COMM SMOVL C00347 BC00347 V=10.0  +MOVJ EC00347
COMM ARCOF
COMM SMOVL C00348 BC00348 V=800.0  +MOVJ EC00348
COMM SMOVL C00349 BC00349 V=1000.0  +MOVJ EC00349
COMM SFTOF3D
COMM 'EndPath W4788
COMM 'Path W4772
COMM SFTOF3D
COMM SFTON3D P041
COMM MOVJ C00350 BC00350 VJ=100.00  +MOVJ EC00350 VJ=100.00
COMM SMOVL C00351 BC00351 V=800.0  +MOVJ EC00351
COMM SMOVL C00352 BC00352 V=150.0 PL=0  +MOVJ EC00352
COMM MACRO1 MJ#(0) ARGF14
COMM ARCON
COMM SMOVL C00353 BC00353 V=10.0  +MOVJ EC00353
COMM SMOVL C00354 BC00354 V=10.0  +MOVJ EC00354
COMM ARCOF
COMM SMOVL C00355 BC00355 V=800.0  +MOVJ EC00355
COMM SMOVL C00356 BC00356 V=1000.0  +MOVJ EC00356
COMM SFTOF3D
COMM 'EndPath W4772
COMM MOVJ C00357 BC00357 VJ=100.00  +MOVJ EC00357 VJ=100.00
COMM '
COMM MOVJ C00358 BC00358 VJ=100.00  +MOVJ EC00358 VJ=100.00
COMM 'Path W4777
COMM SFTOF3D
COMM SFTON3D P040
COMM MOVJ C00359 BC00359 VJ=100.00  +MOVJ EC00359 VJ=100.00
COMM SMOVL C00360 BC00360 V=800.0  +MOVJ EC00360
COMM SMOVL C00361 BC00361 V=150.0 PL=0  +MOVJ EC00361
COMM MACRO1 MJ#(0) ARGF9
COMM ARCON
COMM SMOVL C00362 BC00362 V=10.0  +MOVJ EC00362
COMM SMOVL C00363 BC00363 V=10.0  +MOVJ EC00363
COMM SMOVL C00364 BC00364 V=10.0  +MOVJ EC00364
COMM ARCOF
COMM SMOVL C00365 BC00365 V=800.0  +MOVJ EC00365
COMM SMOVL C00366 BC00366 V=1000.0  +MOVJ EC00366
COMM SFTOF3D
COMM 'EndPath W4777
COMM 'Path W4778
COMM SFTOF3D
COMM SFTON3D P040
COMM MOVJ C00367 BC00367 VJ=100.00  +MOVJ EC00367 VJ=100.00
COMM SMOVL C00368 BC00368 V=800.0  +MOVJ EC00368
COMM SMOVL C00369 BC00369 V=150.0 PL=0  +MOVJ EC00369
COMM MACRO1 MJ#(0) ARGF14
COMM ARCON
COMM SMOVL C00370 BC00370 V=10.0  +MOVJ EC00370
COMM SMOVL C00371 BC00371 V=10.0  +MOVJ EC00371
COMM ARCOF
COMM SMOVL C00372 BC00372 V=800.0  +MOVJ EC00372
COMM SMOVL C00373 BC00373 V=1000.0  +MOVJ EC00373
COMM SFTOF3D
COMM 'EndPath W4778
COMM 'Path W4776
COMM SFTOF3D
COMM SFTON3D P040
COMM MOVJ C00374 BC00374 VJ=100.00  +MOVJ EC00374 VJ=100.00
COMM SMOVL C00375 BC00375 V=800.0  +MOVJ EC00375
COMM SMOVL C00376 BC00376 V=150.0 PL=0  +MOVJ EC00376
COMM ARCON
COMM SMOVL C00377 BC00377 V=10.0  +MOVJ EC00377
COMM SMOVL C00378 BC00378 V=10.0  +MOVJ EC00378
COMM ARCOF
COMM SMOVL C00379 BC00379 V=800.0  +MOVJ EC00379
COMM SMOVL C00380 BC00380 V=1000.0  +MOVJ EC00380
COMM SFTOF3D
COMM 'EndPath W4776
COMM '
COMM MOVJ C00381 BC00381 VJ=100.00  +MOVJ EC00381 VJ=100.00
COMM 'Path W4773
COMM SFTOF3D
COMM SFTON3D P041
COMM MOVJ C00382 BC00382 VJ=100.00  +MOVJ EC00382 VJ=100.00
COMM SMOVL C00383 BC00383 V=800.0  +MOVJ EC00383
COMM SMOVL C00384 BC00384 V=150.0 PL=0  +MOVJ EC00384
COMM ARCON
COMM SMOVL C00385 BC00385 V=9.2  +MOVJ EC00385
COMM ARCOF
COMM SMOVL C00386 BC00386 V=800.0  +MOVJ EC00386
COMM SMOVL C00387 BC00387 V=1000.0  +MOVJ EC00387
COMM SFTOF3D
COMM 'EndPath W4773
COMM '
COMM MOVJ C00388 BC00388 VJ=100.00  +MOVJ EC00388 VJ=100.00
COMM 'Path W4779
COMM SFTOF3D
COMM SFTON3D P040
COMM MOVJ C00389 BC00389 VJ=100.00  +MOVJ EC00389 VJ=100.00
COMM SMOVL C00390 BC00390 V=800.0  +MOVJ EC00390
COMM SMOVL C00391 BC00391 V=150.0 PL=0  +MOVJ EC00391
COMM ARCON
COMM SMOVL C00392 BC00392 V=10.0  +MOVJ EC00392
COMM ARCOF
COMM SMOVL C00393 BC00393 V=800.0  +MOVJ EC00393
COMM SMOVL C00394 BC00394 V=1000.0  +MOVJ EC00394
SFTOF3D
'EndPath W4779
MOVJ C00395 BC00395 VJ=100.00  +MOVJ EC00395 VJ=100.00
'
'
'
'
'uwaga na kolizje-B
'Path W4782
SFTOF3D
SFTON3D P022
MOVJ C00396 BC00396 VJ=30.00  +MOVJ EC00396 VJ=100.00
SMOVL C00397 BC00397 V=800.0  +MOVJ EC00397
'POSPAWANE
SMOVL C00398 BC00398 V=150.0 PL=0  +MOVJ EC00398
MACRO1 MJ#(0) ARGF21
ARCON
SMOVL C00399 BC00399 V=7.5  +MOVJ EC00399
SMOVL C00400 BC00400 V=7.5  +MOVJ EC00400
SMOVL C00401 BC00401 V=7.5  +MOVJ EC00401
ARCOF
SMOVL C00402 BC00402 V=800.0  +MOVJ EC00402
SMOVL C00403 BC00403 V=1000.0  +MOVJ EC00403
SFTOF3D
'Path W4789
SFTOF3D
SFTON3D P022
SMOVL C00404 BC00404 V=666.7  +MOVJ EC00404
SMOVL C00405 BC00405 V=800.0  +MOVJ EC00405
SMOVL C00406 BC00406 V=150.0 PL=0  +MOVJ EC00406
ARCON
SMOVL C00407 BC00407 V=7.5  +MOVJ EC00407
SMOVL C00408 BC00408 V=7.5  +MOVJ EC00408
SMOVL C00409 BC00409 V=7.5  +MOVJ EC00409
ARCOF
SMOVL C00410 BC00410 V=800.0  +MOVJ EC00410
SMOVL C00411 BC00411 V=1000.0  +MOVJ EC00411
SFTOF3D
'EndPath W4789
MOVJ C00412 BC00412 VJ=100.00  +MOVJ EC00412 VJ=100.00
'
MOVJ C00413 BC00413 VJ=15.00  +MOVJ EC00413 VJ=100.00
MOVJ C00414 BC00414 VJ=100.00  +MOVJ EC00414 VJ=100.00
'Path W4784
SFTOF3D
SFTON3D P021
MOVJ C00415 BC00415 VJ=100.00  +MOVJ EC00415 VJ=100.00
SMOVL C00416 BC00416 V=800.0  +MOVJ EC00416
SMOVL C00417 BC00417 V=150.0 PL=0  +MOVJ EC00417
ARCON
SMOVL C00418 BC00418 V=7.5  +MOVJ EC00418
SMOVL C00419 BC00419 V=7.5  +MOVJ EC00419
SMOVL C00420 BC00420 V=7.5  +MOVJ EC00420
ARCOF
SMOVL C00421 BC00421 V=800.0  +MOVJ EC00421
SMOVL C00422 BC00422 V=1000.0  +MOVJ EC00422
SFTOF3D
'EndPath W4784
MOVJ C00423 BC00423 VJ=100.00  +MOVJ EC00423 VJ=100.00
MOVJ C00424 BC00424 VJ=100.00  +MOVJ EC00424 VJ=100.00
'Path W4785
SFTOF3D
SFTON3D P021
MOVJ C00425 BC00425 VJ=100.00  +MOVJ EC00425 VJ=100.00
SMOVL C00426 BC00426 V=800.0  +MOVJ EC00426
SMOVL C00427 BC00427 V=150.0 PL=0  +MOVJ EC00427
ARCON
SMOVL C00428 BC00428 V=7.5  +MOVJ EC00428
SMOVL C00429 BC00429 V=7.5  +MOVJ EC00429
SMOVL C00430 BC00430 V=7.5  +MOVJ EC00430
ARCOF
SMOVL C00431 BC00431 V=800.0  +MOVJ EC00431
SMOVL C00432 BC00432 V=1000.0  +MOVJ EC00432
SFTOF3D
'EndPath W4785
MOVJ C00433 BC00433 VJ=100.00  +MOVJ EC00433 VJ=100.00
'obrot-schodki
MOVJ C00434 BC00434 VJ=100.00  +MOVJ EC00434 VJ=100.00
'Path W4790
SFTOF3D
SFTON3D P031
MOVJ C00435 BC00435 VJ=100.00  +MOVJ EC00435 VJ=100.00
SMOVL C00436 BC00436 V=800.0  +MOVJ EC00436
SMOVL C00437 BC00437 V=150.0 PL=0  +MOVJ EC00437
MACRO1 MJ#(0) ARGF9
ARCON
SMOVL C00438 BC00438 V=8.3  +MOVJ EC00438
SMOVL C00439 BC00439 V=8.3  +MOVJ EC00439
ARCOF
SMOVL C00440 BC00440 V=800.0  +MOVJ EC00440
SMOVL C00441 BC00441 V=1000.0  +MOVJ EC00441
SFTOF3D
'EndPath W4790
'Path W4865
SFTOF3D
SFTON3D P032
MOVJ C00442 BC00442 VJ=100.00  +MOVJ EC00442 VJ=100.00
SMOVL C00443 BC00443 V=800.0  +MOVJ EC00443
SMOVL C00444 BC00444 V=150.0 PL=0  +MOVJ EC00444
ARCON
SMOVL C00445 BC00445 V=8.3  +MOVJ EC00445
SMOVL C00446 BC00446 V=8.3  +MOVJ EC00446
SMOVL C00447 BC00447 V=8.3  +MOVJ EC00447
ARCOF
SMOVL C00448 BC00448 V=800.0  +MOVJ EC00448
SMOVL C00449 BC00449 V=1000.0  +MOVJ EC00449
SFTOF3D
'EndPath W4865
'Path W4866
SFTOF3D
SFTON3D P033
MOVJ C00450 BC00450 VJ=100.00  +MOVJ EC00450 VJ=100.00
SMOVL C00451 BC00451 V=150.0 PL=0  +MOVJ EC00451
ARCON
SMOVL C00452 BC00452 V=8.3  +MOVJ EC00452
ARCOF
SMOVL C00453 BC00453 V=800.0  +MOVJ EC00453
SMOVL C00454 BC00454 V=1000.0  +MOVJ EC00454
SFTOF3D
'EndPath W4866
'
MOVJ C00455 BC00455 VJ=100.00  +MOVJ EC00455 VJ=100.00
'Path W4867
SFTOF3D
SFTON3D P032
MOVJ C00456 BC00456 VJ=100.00  +MOVJ EC00456 VJ=100.00
SMOVL C00457 BC00457 V=800.0  +MOVJ EC00457
SMOVL C00458 BC00458 V=150.0 PL=0  +MOVJ EC00458
MACRO1 MJ#(0) ARGF14
ARCON
SMOVL C00459 BC00459 V=10.0  +MOVJ EC00459
SMOVL C00460 BC00460 V=10.0  +MOVJ EC00460
ARCOF
SMOVL C00461 BC00461 V=800.0  +MOVJ EC00461
SMOVL C00462 BC00462 V=1000.0  +MOVJ EC00462
SFTOF3D
'EndPath W4867
MOVJ C00463 BC00463 VJ=100.00  +MOVJ EC00463 VJ=100.00
'Path W4868
SFTOF3D
SFTON3D P031
MOVJ C00464 BC00464 VJ=100.00  +MOVJ EC00464 VJ=100.00
SMOVL C00465 BC00465 V=800.0  +MOVJ EC00465
SMOVL C00466 BC00466 V=150.0 PL=0  +MOVJ EC00466
ARCON
SMOVL C00467 BC00467 V=10.0  +MOVJ EC00467
SMOVL C00468 BC00468 V=10.0  +MOVJ EC00468
ARCOF
SMOVL C00469 BC00469 V=800.0  +MOVJ EC00469
SMOVL C00470 BC00470 V=1000.0  +MOVJ EC00470
SFTOF3D
'EndPath W4868
MOVJ C00471 BC00471 VJ=100.00  +MOVJ EC00471 VJ=100.00
'
MOVJ C00472 BC00472 VJ=100.00  +MOVJ EC00472 VJ=100.00
MOVJ C00473 BC00473 VJ=100.00  +MOVJ EC00473 VJ=100.00
'Path W4801
SFTOF3D
SFTON3D P034
MOVJ C00474 BC00474 VJ=100.00  +MOVJ EC00474 VJ=100.00
SMOVL C00475 BC00475 V=800.0  +MOVJ EC00475
SMOVL C00476 BC00476 V=150.0 PL=0  +MOVJ EC00476
MACRO1 MJ#(0) ARGF9
ARCON
SMOVL C00477 BC00477 V=8.3  +MOVJ EC00477
SMOVL C00478 BC00478 V=8.3  +MOVJ EC00478
ARCOF
SMOVL C00479 BC00479 V=800.0  +MOVJ EC00479
SMOVL C00480 BC00480 V=1000.0  +MOVJ EC00480
SFTOF3D
'EndPath W4801
'Path W4802
SFTOF3D
SFTON3D P035
MOVJ C00481 BC00481 VJ=100.00  +MOVJ EC00481 VJ=100.00
SMOVL C00482 BC00482 V=800.0  +MOVJ EC00482
SMOVL C00483 BC00483 V=150.0 PL=0  +MOVJ EC00483
ARCON
SMOVL C00484 BC00484 V=8.3  +MOVJ EC00484
SMOVL C00485 BC00485 V=8.3  +MOVJ EC00485
ARCOF
SMOVL C00486 BC00486 V=800.0  +MOVJ EC00486
SMOVL C00487 BC00487 V=1000.0  +MOVJ EC00487
SFTOF3D
'EndPath W4802
'Path W4803
SFTOF3D
SFTON3D P036
MOVJ C00488 BC00488 VJ=100.00  +MOVJ EC00488 VJ=100.00
SMOVL C00489 BC00489 V=800.0  +MOVJ EC00489
SMOVL C00490 BC00490 V=150.0 PL=0  +MOVJ EC00490
ARCON
SMOVL C00491 BC00491 V=8.3  +MOVJ EC00491
SMOVL C00492 BC00492 V=8.3  +MOVJ EC00492
ARCOF
SMOVL C00493 BC00493 V=800.0  +MOVJ EC00493
SMOVL C00494 BC00494 V=1000.0  +MOVJ EC00494
SFTOF3D
'EndPath W4803
'
'Path W4804
SFTOF3D
SFTON3D P035
MOVJ C00495 BC00495 VJ=100.00  +MOVJ EC00495 VJ=100.00
SMOVL C00496 BC00496 V=800.0  +MOVJ EC00496
SMOVL C00497 BC00497 V=150.0 PL=0  +MOVJ EC00497
MACRO1 MJ#(0) ARGF14
ARCON
SMOVL C00498 BC00498 V=10.0  +MOVJ EC00498
SMOVL C00499 BC00499 V=10.0  +MOVJ EC00499
ARCOF
SMOVL C00500 BC00500 V=800.0  +MOVJ EC00500
SMOVL C00501 BC00501 V=1000.0  +MOVJ EC00501
SFTOF3D
'EndPath W4804
'Path W4805
SFTOF3D
SFTON3D P034
MOVJ C00502 BC00502 VJ=100.00  +MOVJ EC00502 VJ=100.00
SMOVL C00503 BC00503 V=800.0  +MOVJ EC00503
SMOVL C00504 BC00504 V=150.0 PL=0  +MOVJ EC00504
ARCON
SMOVL C00505 BC00505 V=10.0  +MOVJ EC00505
SMOVL C00506 BC00506 V=10.0  +MOVJ EC00506
ARCOF
SMOVL C00507 BC00507 V=800.0  +MOVJ EC00507
SMOVL C00508 BC00508 V=1000.0  +MOVJ EC00508
SFTOF3D
COMM MOVL C00509 BC00509 V=1000.0  +MOVJ EC00509 VJ=0.78
COMM MOVL C00510 BC00510 V=1000.0  +MOVJ EC00510 VJ=0.78
COMM MOVL C00511 BC00511 V=1000.0  +MOVJ EC00511 VJ=0.78
COMM PAUSE
COMM SFTOF3D
COMM SFTON3D P041
COMM MOVJ C00512 BC00512 VJ=100.00  +MOVJ EC00512 VJ=100.00
COMM SMOVL C00513 BC00513 V=800.0  +MOVJ EC00513
COMM SMOVL C00514 BC00514 V=150.0 PL=0  +MOVJ EC00514
COMM MACRO1 MJ#(0) ARGF14
COMM ARCON
COMM SMOVL C00515 BC00515 V=13.3  +MOVJ EC00515
COMM SMOVL C00516 BC00516 V=13.3  +MOVJ EC00516
COMM ARCOF
COMM SMOVL C00517 BC00517 V=800.0  +MOVJ EC00517
COMM SMOVL C00518 BC00518 V=1000.0  +MOVJ EC00518
COMM SFTOF3D
COMM 'EndPath W4774
COMM 'Path W4788
COMM SFTOF3D
COMM SFTON3D P041
COMM MOVJ C00519 BC00519 VJ=100.00  +MOVJ EC00519 VJ=100.00
COMM SMOVL C00520 BC00520 V=800.0  +MOVJ EC00520
COMM SMOVL C00521 BC00521 V=150.0 PL=0  +MOVJ EC00521
COMM MACRO1 MJ#(0) ARGF9
COMM ARCON
COMM SMOVL C00522 BC00522 V=15.0  +MOVJ EC00522
COMM SMOVL C00523 BC00523 V=15.0  +MOVJ EC00523
COMM SMOVL C00524 BC00524 V=15.0  +MOVJ EC00524
COMM ARCOF
COMM SMOVL C00525 BC00525 V=800.0  +MOVJ EC00525
COMM SMOVL C00526 BC00526 V=1000.0  +MOVJ EC00526
COMM SFTOF3D
COMM 'EndPath W4788
COMM 'Path W4772
COMM SFTOF3D
COMM SFTON3D P041
COMM MOVJ C00527 BC00527 VJ=100.00  +MOVJ EC00527 VJ=100.00
COMM SMOVL C00528 BC00528 V=800.0  +MOVJ EC00528
COMM SMOVL C00529 BC00529 V=150.0 PL=0  +MOVJ EC00529
COMM MACRO1 MJ#(0) ARGF14
COMM ARCON
COMM SMOVL C00530 BC00530 V=15.0  +MOVJ EC00530
COMM SMOVL C00531 BC00531 V=15.0  +MOVJ EC00531
COMM ARCOF
COMM SMOVL C00532 BC00532 V=800.0  +MOVJ EC00532
COMM SMOVL C00533 BC00533 V=1000.0  +MOVJ EC00533
COMM SFTOF3D
COMM 'EndPath W4772
COMM MOVJ C00534 BC00534 VJ=100.00  +MOVJ EC00534 VJ=100.00
COMM '
COMM MOVJ C00535 BC00535 VJ=100.00  +MOVJ EC00535 VJ=100.00
COMM 'Path W4777
COMM SFTOF3D
COMM SFTON3D P040
COMM MOVJ C00536 BC00536 VJ=100.00  +MOVJ EC00536 VJ=100.00
COMM SMOVL C00537 BC00537 V=800.0  +MOVJ EC00537
COMM SMOVL C00538 BC00538 V=150.0 PL=0  +MOVJ EC00538
COMM MACRO1 MJ#(0) ARGF9
COMM ARCON
COMM SMOVL C00539 BC00539 V=13.3  +MOVJ EC00539
COMM SMOVL C00540 BC00540 V=13.3  +MOVJ EC00540
COMM SMOVL C00541 BC00541 V=13.3  +MOVJ EC00541
COMM ARCOF
COMM SMOVL C00542 BC00542 V=800.0  +MOVJ EC00542
COMM SMOVL C00543 BC00543 V=1000.0  +MOVJ EC00543
COMM SFTOF3D
COMM 'EndPath W4777
COMM 'Path W4778
COMM SFTOF3D
COMM SFTON3D P040
COMM MOVJ C00544 BC00544 VJ=100.00  +MOVJ EC00544 VJ=100.00
COMM SMOVL C00545 BC00545 V=800.0  +MOVJ EC00545
COMM SMOVL C00546 BC00546 V=150.0 PL=0  +MOVJ EC00546
COMM MACRO1 MJ#(0) ARGF14
COMM ARCON
COMM SMOVL C00547 BC00547 V=15.0  +MOVJ EC00547
COMM SMOVL C00548 BC00548 V=15.0  +MOVJ EC00548
COMM ARCOF
COMM SMOVL C00549 BC00549 V=800.0  +MOVJ EC00549
COMM SMOVL C00550 BC00550 V=1000.0  +MOVJ EC00550
COMM SFTOF3D
COMM 'EndPath W4778
COMM 'Path W4776
COMM SFTOF3D
COMM SFTON3D P040
COMM MOVJ C00551 BC00551 VJ=100.00  +MOVJ EC00551 VJ=100.00
COMM SMOVL C00552 BC00552 V=800.0  +MOVJ EC00552
COMM SMOVL C00553 BC00553 V=150.0 PL=0  +MOVJ EC00553
COMM ARCON
COMM SMOVL C00554 BC00554 V=10.0  +MOVJ EC00554
COMM SMOVL C00555 BC00555 V=10.0  +MOVJ EC00555
COMM ARCOF
COMM SMOVL C00556 BC00556 V=800.0  +MOVJ EC00556
COMM SMOVL C00557 BC00557 V=1000.0  +MOVJ EC00557
COMM SFTOF3D
COMM PAUSE
'EndPath W4805
MOVJ C00558 BC00558 VJ=100.00  +MOVJ EC00558 VJ=100.00
'
'
'
MOVJ C00559 BC00559 VJ=100.00  +MOVJ EC00559 VJ=100.00
END
